KUKA KRL program: EPS_2_25748_MH03A_A_20260121065858.src

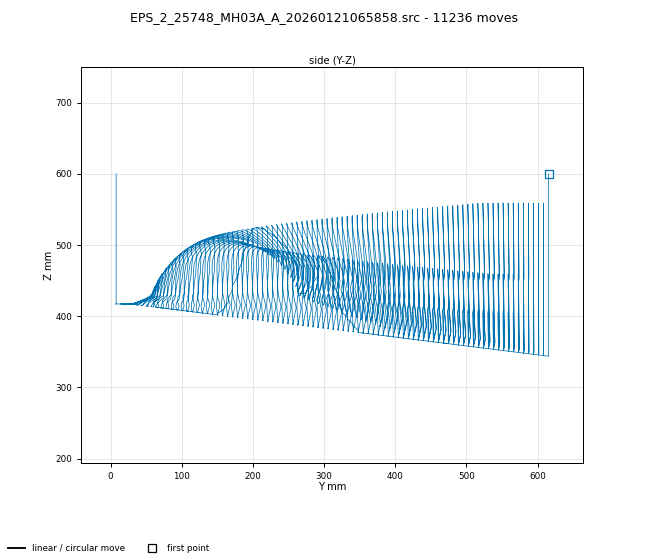
[picture p0: tool path of EPS_2_25748_MH03A_A_20260121065858.src, 11236 of 11238 moves have a stored position in this frame; points joined in program order, loops and branches not executed]
&ACCESS RVP
&REL 4
&COMMENT QRS 19112012
&PARAM EDITMASK = *
DEF PART()
EXT BAS (BAS_COMMAND :IN,REAL :IN )
INT I
BAS (#INITMOV,0 )

;KUKA QRS Post kuka4.cps  Date:22-06-2017 !

File_ID=2998

QRS_PRE_INIT()

;Init var - Until changes are made in qrs_pre_init
Outlet_Square_prg=0
Inlet_1_Square_prg=0
Inlet_2_Square_prg=0
Inlet_3_Square_prg=0
Inlet_4_Square_prg=0
Inlet_5_Square_prg=0

Outlet_1={X 0.000, Y 520.860, Z 458.500, B 0.000, E1 0.000 }
Inlet_1={X 0.000, Y 535.970, Z 408.500, B 0.000, E1 270.000 }
Outlet_1_type=201
Inlet_1_type=101
;QRS#1=Sidecore dimensions
;QRS#2=200-8" PVC SDR 35
;QRS#3=100-4" PVC SDR 28
;QRS#4=
;QRS#5=
;QRS#6=
;QRS#7=
;QRS#8=
;QRS#9=12-08 PSX
;QRS#10=8QRS PSX
;QRS#11=
;QRS#12=
;QRS#13=
;QRS#14=
;QRS#15=
;QRS#16=1220x127x838 2,75'
;QRS#17=EPS Height
;QRS#18=559
;QRS#19=*
;QRS#20= UPDATED VERSION 22-06-2017
;QRS#21=*
Outlet_Square=0100
Inlet_1_Square=045
Inlet_2_Square=0
Inlet_3_Square=0
Inlet_4_Square=0
Inlet_5_Square=0
Mill_Square=1
Outlet_Square_Prg=204
Inlet_1_Square_prg=201

QRS_INIT()

$ADVANCE=5

; T1
PTP {E1 173.608,E2 173.608}
PTP {X 0,Y 615.501,A -85,B 0,C 180,E1 173.608,E2 173.608,E3 0,E4 0,E5 0,E6 0}
QRS_SPEED_INIT()
LIN {X 0,Y 615.501,Z 600,A -85,B 0,C 180,E1 173.608,E2 173.608,E3 0,E4 0,E5 0,E6 0} C_VEL
LIN {X 0,Y 615.501,Z 353.868,A -85,B 0,C 180,E1 173.608,E2 173.608} C_VEL
LIN {X 0,Y 615.501,Z 345.693,A -85,B 0,C 180,E1 173.608,E2 173.608} C_VEL
LIN {X 0,Y 615.488,Z 343.693,A -85,B 0,C 180,E1 173.422,E2 173.422} C_VEL
LIN {X 0,Y 615.492,Z 343.688,A -85,B 0,C 180,E1 170.801,E2 170.801} C_VEL
LIN {X 0,Y 615.492,Z 343.699,A -85,B 0,C 180,E1 168.139,E2 168.139} C_VEL
LIN {X 0,Y 615.481,Z 343.69,A -85,B 0,C 180,E1 165.451,E2 165.451} C_VEL
LIN {X 0,Y 615.493,Z 343.692,A -85,B 0,C 180,E1 162.73,E2 162.73} C_VEL
LIN {X 0,Y 615.49,Z 343.695,A -85,B 0,C 180,E1 159.967,E2 159.967} C_VEL
LIN {X 0,Y 615.481,Z 343.69,A -85,B 0,C 180,E1 157.155,E2 157.155} C_VEL
LIN {X 0,Y 615.482,Z 343.693,A -85,B 0,C 180,E1 154.284,E2 154.284} C_VEL
LIN {X 0,Y 615.479,Z 343.699,A -85,B 0,C 180,E1 151.551,E2 151.551} C_VEL
LIN {X 0,Y 615.485,Z 343.689,A -85,B 0,C 180,E1 148.915,E2 148.915} C_VEL
LIN {X 0,Y 615.49,Z 343.692,A -85,B 0,C 180,E1 145.978,E2 145.978} C_VEL
LIN {X 0,Y 615.487,Z 343.702,A -85,B 0,C 180,E1 143.063,E2 143.063} C_VEL
LIN {X 0,Y 615.49,Z 343.689,A -85,B 0,C 180,E1 140.25,E2 140.25} C_VEL
LIN {X 0,Y 615.485,Z 343.693,A -85,B 0,C 180,E1 137.647,E2 137.647} C_VEL
LIN {X 0,Y 615.491,Z 343.694,A -85,B 0,C 180,E1 134.932,E2 134.932} C_VEL
LIN {X 0,Y 615.485,Z 343.689,A -85,B 0,C 180,E1 132.08,E2 132.08} C_VEL
LIN {X 0,Y 615.489,Z 343.7,A -85,B 0,C 180,E1 129.75,E2 129.75} C_VEL
LIN {X 0,Y 615.476,Z 343.692,A -85,B 0,C 180,E1 126.935,E2 126.935} C_VEL
LIN {X 0,Y 615.492,Z 343.701,A -85,B 0,C 180,E1 124.701,E2 124.701} C_VEL
LIN {X 0,Y 615.49,Z 343.688,A -85,B 0,C 180,E1 122.331,E2 122.331} C_VEL
LIN {X 0,Y 615.492,Z 343.695,A -85,B 0,C 180,E1 119.406,E2 119.406} C_VEL
LIN {X 0,Y 615.476,Z 343.691,A -85,B 0,C 180,E1 117.042,E2 117.042} C_VEL
LIN {X 0,Y 615.48,Z 343.694,A -85,B 0,C 180,E1 114.272,E2 114.272} C_VEL
LIN {X 0,Y 615.496,Z 343.697,A -85,B 0,C 180,E1 111.431,E2 111.431} C_VEL
LIN {X 0,Y 615.488,Z 343.689,A -85,B 0,C 180,E1 108.604,E2 108.604} C_VEL
LIN {X 0,Y 615.492,Z 343.691,A -85,B 0,C 180,E1 105.905,E2 105.905} C_VEL
LIN {X 0,Y 615.485,Z 343.696,A -85,B 0,C 180,E1 103.201,E2 103.201} C_VEL
LIN {X 0,Y 615.481,Z 343.69,A -85,B 0,C 180,E1 100.527,E2 100.527} C_VEL
LIN {X 0,Y 615.487,Z 343.701,A -85,B 0,C 180,E1 97.876,E2 97.876} C_VEL
LIN {X 0,Y 615.48,Z 343.691,A -85,B 0,C 180,E1 95.241,E2 95.241} C_VEL
LIN {X 0,Y 615.48,Z 343.695,A -85,B 0,C 180,E1 92.618,E2 92.618} C_VEL
LIN {X 0,Y 615.49,Z 343.692,A -85,B 0,C 180,E1 90,E2 90} C_VEL
LIN {X 0,Y 615.48,Z 343.692,A -85,B 0,C 180,E1 87.382,E2 87.382} C_VEL
LIN {X 0,Y 615.486,Z 343.698,A -85,B 0,C 180,E1 84.759,E2 84.759} C_VEL
LIN {X 0,Y 615.488,Z 343.688,A -85,B 0,C 180,E1 82.124,E2 82.124} C_VEL
LIN {X 0,Y 615.497,Z 343.697,A -85,B 0,C 180,E1 79.473,E2 79.473} C_VEL
LIN {X 0,Y 615.479,Z 343.692,A -85,B 0,C 180,E1 76.798,E2 76.798} C_VEL
LIN {X 0,Y 615.485,Z 343.691,A -85,B 0,C 180,E1 74.095,E2 74.095} C_VEL
LIN {X 0,Y 615.488,Z 343.699,A -85,B 0,C 180,E1 71.354,E2 71.354} C_VEL
LIN {X 0,Y 615.485,Z 343.689,A -85,B 0,C 180,E1 68.568,E2 68.568} C_VEL
LIN {X 0,Y 615.482,Z 343.692,A -85,B 0,C 180,E1 65.728,E2 65.728} C_VEL
LIN {X 0,Y 615.492,Z 343.7,A -85,B 0,C 180,E1 62.955,E2 62.955} C_VEL
LIN {X 0,Y 615.482,Z 343.69,A -85,B 0,C 180,E1 60.207,E2 60.207} C_VEL
LIN {X 0,Y 615.495,Z 343.692,A -85,B 0,C 180,E1 57.543,E2 57.543} C_VEL
LIN {X 0,Y 615.478,Z 343.691,A -85,B 0,C 180,E1 55.184,E2 55.184} C_VEL
LIN {X 0,Y 615.497,Z 343.697,A -85,B 0,C 180,E1 52.758,E2 52.758} C_VEL
LIN {X 0,Y 615.482,Z 343.694,A -85,B 0,C 180,E1 49.912,E2 49.912} C_VEL
LIN {X 0,Y 615.495,Z 343.695,A -85,B 0,C 180,E1 47.647,E2 47.647} C_VEL
LIN {X 0,Y 615.482,Z 343.693,A -85,B 0,C 180,E1 44.931,E2 44.931} C_VEL
LIN {X 0,Y 615.482,Z 343.69,A -85,B 0,C 180,E1 42.079,E2 42.079} C_VEL
LIN {X 0,Y 615.496,Z 343.694,A -85,B 0,C 180,E1 39.75,E2 39.75} C_VEL
LIN {X 0,Y 615.486,Z 343.689,A -85,B 0,C 180,E1 36.936,E2 36.936} C_VEL
LIN {X 0,Y 615.487,Z 343.691,A -85,B 0,C 180,E1 34.022,E2 34.022} C_VEL
LIN {X 0,Y 615.49,Z 343.699,A -85,B 0,C 180,E1 31.086,E2 31.086} C_VEL
LIN {X 0,Y 615.489,Z 343.835,A -85,B 0,C 180,E1 29.697,E2 29.697} C_VEL
LIN {X 0,Y 615.498,Z 350.25,A -85,B 0,C 180,E1 27.046,E2 27.046} C_VEL
LIN {X 0,Y 615.488,Z 357.77,A -85,B 0,C 180,E1 24.008,E2 24.008} C_VEL
LIN {X 0,Y 615.478,Z 364.29,A -85,B 0,C 180,E1 21.432,E2 21.432} C_VEL
LIN {X 0,Y 615.476,Z 371.461,A -85,B 0,C 180,E1 18.646,E2 18.646} C_VEL
LIN {X 0,Y 615.488,Z 378.635,A -85,B 0,C 180,E1 15.905,E2 15.905} C_VEL
LIN {X 0,Y 615.494,Z 385.799,A -85,B 0,C 180,E1 13.201,E2 13.201} C_VEL
LIN {X 0,Y 615.486,Z 392.972,A -85,B 0,C 180,E1 10.527,E2 10.527} C_VEL
LIN {X 0,Y 615.478,Z 400.129,A -85,B 0,C 180,E1 7.876,E2 7.876} C_VEL
LIN {X 0,Y 615.487,Z 403.222,A -85,B 0,C 180,E1 6.737,E2 6.737} C_VEL
LIN {X 0,Y 615.489,Z 413.526,A -85,B 0,C 180,E1 6.392,E2 6.392} C_VEL
LIN {X 0,Y 615.478,Z 421.945,A -85,B 0,C 180,E1 5.981,E2 5.981} C_VEL
LIN {X 0,Y 615.487,Z 429.67,A -85,B 0,C 180,E1 5.488,E2 5.488} C_VEL
LIN {X 0,Y 615.489,Z 436.516,A -85,B 0,C 180,E1 4.913,E2 4.913} C_VEL
LIN {X 0,Y 615.497,Z 442.667,A -85,B 0,C 180,E1 4.256,E2 4.256} C_VEL
LIN {X 0,Y 615.497,Z 447.515,A -85,B 0,C 180,E1 3.601,E2 3.601} C_VEL
LIN {X 0,Y 615.496,Z 451.25,A -85,B 0,C 180,E1 2.945,E2 2.945} C_VEL
LIN {X 0,Y 615.498,Z 455.229,A -85,B 0,C 180,E1 1.963,E2 1.963} C_VEL
LIN {X 0,Y 615.497,Z 456.963,A -85,B 0,C 180,E1 1.309,E2 1.309} C_VEL
LIN {X 0,Y 615.496,Z 458.004,A -85,B 0,C 180,E1 0.654,E2 0.654} C_VEL
LIN {X 0,Y 615.494,Z 458.384,A -85,B 0,C 180,E1 0,E2 0} C_VEL
LIN {X 0,Y 615.496,Z 458.105,A -85,B 0,C 180,E1 -0.654,E2 -0.654} C_VEL
LIN {X 0,Y 615.497,Z 457.166,A -85,B 0,C 180,E1 -1.309,E2 -1.309} C_VEL
LIN {X 0,Y 615.496,Z 455.536,A -85,B 0,C 180,E1 -1.963,E2 -1.963} C_VEL
LIN {X 0,Y 615.498,Z 451.663,A -85,B 0,C 180,E1 -2.945,E2 -2.945} C_VEL
LIN {X 0,Y 615.5,Z 447.012,A -85,B 0,C 180,E1 -3.764,E2 -3.764} C_VEL
LIN {X 0,Y 615.498,Z 442.03,A -85,B 0,C 180,E1 -4.42,E2 -4.42} C_VEL
LIN {X 0,Y 615.482,Z 435.756,A -85,B 0,C 180,E1 -5.077,E2 -5.077} C_VEL
LIN {X 0,Y 615.483,Z 428.589,A -85,B 0,C 180,E1 -5.652,E2 -5.652} C_VEL
LIN {X 0,Y 615.483,Z 420.605,A -85,B 0,C 180,E1 -6.145,E2 -6.145} C_VEL
LIN {X 0,Y 615.492,Z 411.022,A -85,B 0,C 180,E1 -6.579,E2 -6.579} C_VEL
LIN {X 0,Y 615.48,Z 403.195,A -85,B 0,C 180,E1 -6.838,E2 -6.838} C_VEL
LIN {X 0,Y 615.489,Z 396.799,A -85,B 0,C 180,E1 -9.199,E2 -9.199} C_VEL
LIN {X 0,Y 615.477,Z 389.625,A -85,B 0,C 180,E1 -11.861,E2 -11.861} C_VEL
LIN {X 0,Y 615.481,Z 382.466,A -85,B 0,C 180,E1 -14.549,E2 -14.549} C_VEL
LIN {X 0,Y 615.492,Z 375.279,A -85,B 0,C 180,E1 -17.27,E2 -17.27} C_VEL
LIN {X 0,Y 615.493,Z 368.112,A -85,B 0,C 180,E1 -20.033,E2 -20.033} C_VEL
LIN {X 0,Y 615.482,Z 360.924,A -85,B 0,C 180,E1 -22.845,E2 -22.845} C_VEL
LIN {X 0,Y 615.476,Z 354.12,A -85,B 0,C 180,E1 -25.566,E2 -25.566} C_VEL
LIN {X 0,Y 615.485,Z 348.349,A -85,B 0,C 180,E1 -27.915,E2 -27.915} C_VEL
LIN {X 0,Y 615.494,Z 343.696,A -85,B 0,C 180,E1 -29.886,E2 -29.886} C_VEL
LIN {X 0,Y 615.487,Z 343.699,A -85,B 0,C 180,E1 -32.458,E2 -32.458} C_VEL
LIN {X 0,Y 615.498,Z 343.7,A -85,B 0,C 180,E1 -34.815,E2 -34.815} C_VEL
LIN {X 0,Y 615.481,Z 343.699,A -85,B 0,C 180,E1 -37.243,E2 -37.243} C_VEL
LIN {X 0,Y 615.497,Z 343.7,A -85,B 0,C 180,E1 -40.09,E2 -40.09} C_VEL
LIN {X 0,Y 615.491,Z 343.699,A -85,B 0,C 180,E1 -43.047,E2 -43.047} C_VEL
LIN {X 0,Y 615.491,Z 343.697,A -85,B 0,C 180,E1 -46.002,E2 -46.002} C_VEL
LIN {X 0,Y 615.497,Z 343.7,A -85,B 0,C 180,E1 -48.527,E2 -48.527} C_VEL
LIN {X 0,Y 615.478,Z 343.699,A -85,B 0,C 180,E1 -51.095,E2 -51.095} C_VEL
LIN {X 0,Y 615.491,Z 343.699,A -85,B 0,C 180,E1 -53.575,E2 -53.575} C_VEL
LIN {X 0,Y 615.493,Z 343.696,A -85,B 0,C 180,E1 -56.465,E2 -56.465} C_VEL
LIN {X 0,Y 615.491,Z 343.7,A -85,B 0,C 180,E1 -59.08,E2 -59.08} C_VEL
LIN {X 0,Y 615.494,Z 343.696,A -85,B 0,C 180,E1 -61.549,E2 -61.549} C_VEL
LIN {X 0,Y 615.488,Z 343.839,A -85,B 0,C 180,E1 -62.593,E2 -62.593} C_VEL
LIN {X 0,Y 615.489,Z 361.436,A -85,B 0,C 180,E1 -65.369,E2 -65.369} C_VEL
LIN {X 0,Y 615.488,Z 379.892,A -85,B 0,C 180,E1 -68.216,E2 -68.216} C_VEL
LIN {X 0,Y 615.492,Z 398.326,A -85,B 0,C 180,E1 -71.008,E2 -71.008} C_VEL
LIN {X 0,Y 615.493,Z 417.271,A -85,B 0,C 180,E1 -73.832,E2 -73.832} C_VEL
LIN {X 0,Y 615.478,Z 436.29,A -85,B 0,C 180,E1 -76.63,E2 -76.63} C_VEL
LIN {X 0,Y 615.497,Z 447.777,A -85,B 0,C 180,E1 -78.306,E2 -78.306} C_VEL
LIN {X 0,Y 615.483,Z 462.234,A -85,B 0,C 180,E1 -78.556,E2 -78.556} C_VEL
LIN {X 0,Y 615.481,Z 475.31,A -85,B 0,C 180,E1 -78.921,E2 -78.921} C_VEL
LIN {X 0,Y 615.489,Z 487.115,A -85,B 0,C 180,E1 -79.383,E2 -79.383} C_VEL
LIN {X 0,Y 615.487,Z 498.572,A -85,B 0,C 180,E1 -79.972,E2 -79.972} C_VEL
LIN {X 0,Y 615.499,Z 510.019,A -85,B 0,C 180,E1 -80.718,E2 -80.718} C_VEL
LIN {X 0,Y 615.498,Z 519.255,A -85,B 0,C 180,E1 -81.463,E2 -81.463} C_VEL
LIN {X 0,Y 615.499,Z 527.652,A -85,B 0,C 180,E1 -82.289,E2 -82.289} C_VEL
LIN {X 0,Y 615.497,Z 535.69,A -85,B 0,C 180,E1 -83.259,E2 -83.259} C_VEL
LIN {X 0,Y 615.499,Z 541.422,A -85,B 0,C 180,E1 -84.101,E2 -84.101} C_VEL
LIN {X 0,Y 615.496,Z 546.872,A -85,B 0,C 180,E1 -85.087,E2 -85.087} C_VEL
LIN {X 0,Y 615.496,Z 551.14,A -85,B 0,C 180,E1 -86.071,E2 -86.071} C_VEL
LIN {X 0,Y 615.495,Z 553.398,A -85,B 0,C 180,E1 -86.727,E2 -86.727} C_VEL
LIN {X 0,Y 615.497,Z 555.233,A -85,B 0,C 180,E1 -87.382,E2 -87.382} C_VEL
LIN {X 0,Y 615.499,Z 556.607,A -85,B 0,C 180,E1 -88.037,E2 -88.037} C_VEL
LIN {X 0,Y 615.496,Z 558.173,A -85,B 0,C 180,E1 -89.346,E2 -89.346} C_VEL
LIN {X 0,Y 615.494,Z 558.389,A -85,B 0,C 180,E1 -90,E2 -90} C_VEL
LIN {X 0,Y 615.496,Z 557.58,A -85,B 0,C 180,E1 -91.308,E2 -91.308} C_VEL
LIN {X 0,Y 615.499,Z 556.608,A -85,B 0,C 180,E1 -91.963,E2 -91.963} C_VEL
LIN {X 0,Y 615.497,Z 555.233,A -85,B 0,C 180,E1 -92.618,E2 -92.618} C_VEL
LIN {X 0,Y 615.496,Z 552.35,A -85,B 0,C 180,E1 -93.601,E2 -93.601} C_VEL
LIN {X 0,Y 615.498,Z 548.442,A -85,B 0,C 180,E1 -94.584,E2 -94.584} C_VEL
LIN {X 0,Y 615.499,Z 543.405,A -85,B 0,C 180,E1 -95.57,E2 -95.57} C_VEL
LIN {X 0,Y 615.497,Z 536.87,A -85,B 0,C 180,E1 -96.583,E2 -96.583} C_VEL
LIN {X 0,Y 615.497,Z 529.134,A -85,B 0,C 180,E1 -97.545,E2 -97.545} C_VEL
LIN {X 0,Y 615.498,Z 521.046,A -85,B 0,C 180,E1 -98.371,E2 -98.371} C_VEL
LIN {X 0,Y 615.499,Z 511.169,A -85,B 0,C 180,E1 -99.199,E2 -99.199} C_VEL
LIN {X 0,Y 615.492,Z 499.982,A -85,B 0,C 180,E1 -99.945,E2 -99.945} C_VEL
LIN {X 0,Y 615.484,Z 489.025,A -85,B 0,C 180,E1 -100.527,E2 -100.527} C_VEL
LIN {X 0,Y 615.482,Z 476.477,A -85,B 0,C 180,E1 -101.041,E2 -101.041} C_VEL
LIN {X 0,Y 615.481,Z 464.07,A -85,B 0,C 180,E1 -101.402,E2 -101.402} C_VEL
LIN {X 0,Y 615.495,Z 450.47,A -85,B 0,C 180,E1 -101.652,E2 -101.652} C_VEL
LIN {X 0,Y 615.497,Z 447.778,A -85,B 0,C 180,E1 -101.693,E2 -101.693} C_VEL
LIN {X 0,Y 615.494,Z 427.094,A -85,B 0,C 180,E1 -104.718,E2 -104.718} C_VEL
LIN {X 0,Y 615.492,Z 407.539,A -85,B 0,C 180,E1 -107.613,E2 -107.613} C_VEL
LIN {X 0,Y 615.487,Z 389.682,A -85,B 0,C 180,E1 -110.295,E2 -110.295} C_VEL
LIN {X 0,Y 615.479,Z 371.822,A -85,B 0,C 180,E1 -113.022,E2 -113.022} C_VEL
LIN {X 0,Y 615.5,Z 354.515,A -85,B 0,C 180,E1 -115.715,E2 -115.715} C_VEL
LIN {X 0,Y 615.489,Z 343.689,A -85,B 0,C 180,E1 -117.453,E2 -117.453} C_VEL
LIN {X 0,Y 615.5,Z 343.7,A -85,B 0,C 180,E1 -120.159,E2 -120.159} C_VEL
LIN {X 0,Y 615.494,Z 343.688,A -85,B 0,C 180,E1 -122.457,E2 -122.457} C_VEL
LIN {X 0,Y 615.487,Z 343.693,A -85,B 0,C 180,E1 -124.815,E2 -124.815} C_VEL
LIN {X 0,Y 615.487,Z 343.692,A -85,B 0,C 180,E1 -127.242,E2 -127.242} C_VEL
LIN {X 0,Y 615.492,Z 343.699,A -85,B 0,C 180,E1 -130.089,E2 -130.089} C_VEL
LIN {X 0,Y 615.495,Z 343.689,A -85,B 0,C 180,E1 -132.352,E2 -132.352} C_VEL
LIN {X 0,Y 615.489,Z 343.699,A -85,B 0,C 180,E1 -135.068,E2 -135.068} C_VEL
LIN {X 0,Y 615.482,Z 343.691,A -85,B 0,C 180,E1 -137.92,E2 -137.92} C_VEL
LIN {X 0,Y 615.491,Z 343.7,A -85,B 0,C 180,E1 -140.25,E2 -140.25} C_VEL
LIN {X 0,Y 615.488,Z 343.691,A -85,B 0,C 180,E1 -143.063,E2 -143.063} C_VEL
LIN {X 0,Y 615.489,Z 343.688,A -85,B 0,C 180,E1 -145.978,E2 -145.978} C_VEL
LIN {X 0,Y 615.482,Z 343.694,A -85,B 0,C 180,E1 -148.915,E2 -148.915} C_VEL
LIN {X 0,Y 615.48,Z 343.695,A -85,B 0,C 180,E1 -151.551,E2 -151.551} C_VEL
LIN {X 0,Y 615.478,Z 343.69,A -85,B 0,C 180,E1 -154.284,E2 -154.284} C_VEL
LIN {X 0,Y 615.476,Z 343.694,A -85,B 0,C 180,E1 -156.443,E2 -156.443} C_VEL
LIN {X 0,Y 615.499,Z 343.699,A -85,B 0,C 180,E1 -158.568,E2 -158.568} C_VEL
LIN {X 0,Y 615.477,Z 343.693,A -85,B 0,C 180,E1 -161.398,E2 -161.398} C_VEL
LIN {X 0,Y 615.478,Z 343.692,A -85,B 0,C 180,E1 -164.095,E2 -164.095} C_VEL
LIN {X 0,Y 615.498,Z 343.697,A -85,B 0,C 180,E1 -166.799,E2 -166.799} C_VEL
LIN {X 0,Y 615.486,Z 343.689,A -85,B 0,C 180,E1 -169.473,E2 -169.473} C_VEL
LIN {X 0,Y 615.484,Z 343.697,A -85,B 0,C 180,E1 -172.124,E2 -172.124} C_VEL
LIN {X 0,Y 615.487,Z 343.691,A -85,B 0,C 180,E1 -174.759,E2 -174.759} C_VEL
LIN {X 0,Y 615.492,Z 343.69,A -85,B 0,C 180,E1 -177.382,E2 -177.382} C_VEL
LIN {X 0,Y 615.489,Z 343.695,A -85,B 0,C 180,E1 -180,E2 -180} C_VEL
LIN {X 0,Y 615.488,Z 343.688,A -85,B 0,C 180,E1 -182.618,E2 -182.618} C_VEL
LIN {X 0,Y 615.496,Z 343.7,A -85,B 0,C 180,E1 -185.241,E2 -185.241} C_VEL
LIN {X 0,Y 615.488,Z 343.693,A -85,B 0,C 180,E1 -186.578,E2 -186.578} C_VEL
LIN {X 0,Y 614.817,Z 343.842,A -85,B 0,C 180,E1 -187.124,E2 -187.124} C_VEL
LIN {X 0,Y 611.986,Z 344.251,A -85,B 0,C 180,E1 -188.01,E2 -188.01} C_VEL
LIN {X 0,Y 609.592,Z 344.56,A -85,B 0,C 180,E1 -188.723,E2 -188.723} C_VEL
LIN {X 0,Y 608.553,Z 344.679,A -85,B 0,C 180,E1 -189.272,E2 -189.272} C_VEL
LIN {X 0,Y 608.461,Z 344.689,A -85,B 0,C 180,E1 -189.459,E2 -189.459} C_VEL
LIN {X 0,Y 608.466,Z 344.696,A -85,B 0,C 180,E1 -192,E2 -192} C_VEL
LIN {X 0,Y 608.472,Z 344.689,A -85,B 0,C 180,E1 -194.721,E2 -194.721} C_VEL
LIN {X 0,Y 608.456,Z 344.691,A -85,B 0,C 180,E1 -197.477,E2 -197.477} C_VEL
LIN {X 0,Y 608.464,Z 344.697,A -85,B 0,C 180,E1 -200.274,E2 -200.274} C_VEL
LIN {X 0,Y 608.46,Z 344.691,A -85,B 0,C 180,E1 -202.476,E2 -202.476} C_VEL
LIN {X 0,Y 608.457,Z 344.69,A -85,B 0,C 180,E1 -204.571,E2 -204.571} C_VEL
LIN {X 0,Y 608.484,Z 344.69,A -85,B 0,C 180,E1 -207.208,E2 -207.208} C_VEL
LIN {X 0,Y 608.47,Z 344.691,A -85,B 0,C 180,E1 -209.972,E2 -209.972} C_VEL
LIN {X 0,Y 608.455,Z 344.69,A -85,B 0,C 180,E1 -212.88,E2 -212.88} C_VEL
LIN {X 0,Y 608.443,Z 344.699,A -85,B 0,C 180,E1 -215.278,E2 -215.278} C_VEL
LIN {X 0,Y 608.466,Z 344.689,A -85,B 0,C 180,E1 -217.747,E2 -217.747} C_VEL
LIN {X 0,Y 608.453,Z 344.698,A -85,B 0,C 180,E1 -220.329,E2 -220.329} C_VEL
LIN {X 0,Y 608.452,Z 344.691,A -85,B 0,C 180,E1 -222.96,E2 -222.96} C_VEL
LIN {X 0,Y 608.46,Z 344.692,A -85,B 0,C 180,E1 -225.736,E2 -225.736} C_VEL
LIN {X 0,Y 608.462,Z 344.697,A -85,B 0,C 180,E1 -228.658,E2 -228.658} C_VEL
LIN {X 0,Y 608.471,Z 344.692,A -85,B 0,C 180,E1 -231.76,E2 -231.76} C_VEL
LIN {X 0,Y 608.448,Z 344.695,A -85,B 0,C 180,E1 -233.955,E2 -233.955} C_VEL
LIN {X 0,Y 608.465,Z 344.689,A -85,B 0,C 180,E1 -236.329,E2 -236.329} C_VEL
LIN {X 0,Y 608.449,Z 344.698,A -85,B 0,C 180,E1 -238.733,E2 -238.733} C_VEL
LIN {X 0,Y 608.473,Z 344.688,A -85,B 0,C 180,E1 -241.38,E2 -241.38} C_VEL
LIN {X 0,Y 608.478,Z 344.688,A -85,B 0,C 180,E1 -244.278,E2 -244.278} C_VEL
LIN {X 0,Y 608.455,Z 344.696,A -85,B 0,C 180,E1 -246.876,E2 -246.876} C_VEL
LIN {X 0,Y 608.468,Z 344.689,A -85,B 0,C 180,E1 -249.322,E2 -249.322} C_VEL
LIN {X 0,Y 608.456,Z 344.695,A -85,B 0,C 180,E1 -251.828,E2 -251.828} C_VEL
LIN {X 0,Y 608.467,Z 344.689,A -85,B 0,C 180,E1 -254.594,E2 -254.594} C_VEL
LIN {X 0,Y 608.473,Z 344.691,A -85,B 0,C 180,E1 -257.323,E2 -257.323} C_VEL
LIN {X 0,Y 608.465,Z 344.692,A -85,B 0,C 180,E1 -260.023,E2 -260.023} C_VEL
LIN {X 0,Y 608.462,Z 344.69,A -85,B 0,C 180,E1 -262.701,E2 -262.701} C_VEL
LIN {X 0,Y 608.464,Z 344.697,A -85,B 0,C 180,E1 -265.363,E2 -265.363} C_VEL
LIN {X 0,Y 608.469,Z 344.689,A -85,B 0,C 180,E1 -268.014,E2 -268.014} C_VEL
LIN {X 0,Y 608.48,Z 344.691,A -85,B 0,C 180,E1 -270.662,E2 -270.662} C_VEL
LIN {X 0,Y 608.475,Z 344.69,A -85,B 0,C 180,E1 -273.311,E2 -273.311} C_VEL
LIN {X 0,Y 608.492,Z 344.686,A -85,B 0,C 180,E1 -275.967,E2 -275.967} C_VEL
LIN {X 0,Y 608.457,Z 344.696,A -85,B 0,C 180,E1 -278.636,E2 -278.636} C_VEL
LIN {X 0,Y 608.459,Z 344.69,A -85,B 0,C 180,E1 -281.324,E2 -281.324} C_VEL
LIN {X 0,Y 608.473,Z 344.691,A -85,B 0,C 180,E1 -284.038,E2 -284.038} C_VEL
LIN {X 0,Y 608.479,Z 344.69,A -85,B 0,C 180,E1 -286.783,E2 -286.783} C_VEL
LIN {X 0,Y 608.45,Z 344.691,A -85,B 0,C 180,E1 -289.571,E2 -289.571} C_VEL
LIN {X 0,Y 608.481,Z 344.69,A -85,B 0,C 180,E1 -292.405,E2 -292.405} C_VEL
LIN {X 0,Y 608.454,Z 344.696,A -85,B 0,C 180,E1 -295.301,E2 -295.301} C_VEL
LIN {X 0,Y 608.451,Z 344.693,A -85,B 0,C 180,E1 -297.518,E2 -297.518} C_VEL
LIN {X 0,Y 608.463,Z 344.691,A -85,B 0,C 180,E1 -299.97,E2 -299.97} C_VEL
LIN {X 0,Y 608.461,Z 344.689,A -85,B 0,C 180,E1 -302.88,E2 -302.88} C_VEL
LIN {X 0,Y 608.44,Z 344.697,A -85,B 0,C 180,E1 -305.278,E2 -305.278} C_VEL
LIN {X 0,Y 608.469,Z 344.689,A -85,B 0,C 180,E1 -307.747,E2 -307.747} C_VEL
LIN {X 0,Y 608.451,Z 344.696,A -85,B 0,C 180,E1 -310.329,E2 -310.329} C_VEL
LIN {X 0,Y 608.452,Z 344.691,A -85,B 0,C 180,E1 -312.96,E2 -312.96} C_VEL
LIN {X 0,Y 608.45,Z 344.695,A -85,B 0,C 180,E1 -315.737,E2 -315.737} C_VEL
LIN {X 0,Y 608.46,Z 344.695,A -85,B 0,C 180,E1 -318.658,E2 -318.658} C_VEL
LIN {X 0,Y 608.472,Z 344.688,A -85,B 0,C 180,E1 -321.412,E2 -321.412} C_VEL
LIN {X 0,Y 608.482,Z 344.693,A -85,B 0,C 180,E1 -323.95,E2 -323.95} C_VEL
LIN {X 0,Y 608.448,Z 344.691,A -85,B 0,C 180,E1 -326.328,E2 -326.328} C_VEL
LIN {X 0,Y 608.465,Z 344.695,A -85,B 0,C 180,E1 -328.73,E2 -328.73} C_VEL
LIN {X 0,Y 608.481,Z 344.879,A -85,B 0,C 180,E1 -330.316,E2 -330.316} C_VEL
LIN {X 0,Y 608.446,Z 351.891,A -85,B 0,C 180,E1 -333.225,E2 -333.225} C_VEL
LIN {X 0,Y 608.457,Z 358.354,A -85,B 0,C 180,E1 -335.853,E2 -335.853} C_VEL
LIN {X 0,Y 608.442,Z 364.518,A -85,B 0,C 180,E1 -338.307,E2 -338.307} C_VEL
LIN {X 0,Y 608.431,Z 371.734,A -85,B 0,C 180,E1 -341.13,E2 -341.13} C_VEL
LIN {X 0,Y 608.446,Z 378.949,A -85,B 0,C 180,E1 -343.906,E2 -343.906} C_VEL
LIN {X 0,Y 608.437,Z 386.166,A -85,B 0,C 180,E1 -346.643,E2 -346.643} C_VEL
LIN {X 0,Y 608.424,Z 393.382,A -85,B 0,C 180,E1 -349.349,E2 -349.349} C_VEL
LIN {X 0,Y 608.41,Z 400.599,A -85,B 0,C 180,E1 -352.032,E2 -352.032} C_VEL
LIN {X 0,Y 608.433,Z 403.853,A -85,B 0,C 180,E1 -353.186,E2 -353.186} C_VEL
LIN {X 0,Y 608.478,Z 414.079,A -85,B 0,C 180,E1 -353.534,E2 -353.534} C_VEL
LIN {X 0,Y 608.454,Z 422.472,A -85,B 0,C 180,E1 -353.95,E2 -353.95} C_VEL
LIN {X 0,Y 608.453,Z 431.252,A -85,B 0,C 180,E1 -354.532,E2 -354.532} C_VEL
LIN {X 0,Y 608.448,Z 437.027,A -85,B 0,C 180,E1 -355.03,E2 -355.03} C_VEL
LIN {X 0,Y 608.443,Z 443.205,A -85,B 0,C 180,E1 -355.694,E2 -355.694} C_VEL
LIN {X 0,Y 608.451,Z 448.067,A -85,B 0,C 180,E1 -356.358,E2 -356.358} C_VEL
LIN {X 0,Y 608.451,Z 451.818,A -85,B 0,C 180,E1 -357.021,E2 -357.021} C_VEL
LIN {X 0,Y 608.443,Z 455.825,A -85,B 0,C 180,E1 -358.014,E2 -358.014} C_VEL
LIN {X 0,Y 608.449,Z 457.568,A -85,B 0,C 180,E1 -358.676,E2 -358.676} C_VEL
LIN {X 0,Y 608.439,Z 458.615,A -85,B 0,C 180,E1 -359.338,E2 -359.338} C_VEL
LIN {X 0,Y 608.434,Z 458.995,A -85,B 0,C 180,E1 -360,E2 -360} C_VEL
LIN {X 0,Y 608.439,Z 458.714,A -85,B 0,C 180,E1 -360.662,E2 -360.662} C_VEL
LIN {X 0,Y 608.449,Z 457.768,A -85,B 0,C 180,E1 -361.324,E2 -361.324} C_VEL
LIN {X 0,Y 608.442,Z 456.128,A -85,B 0,C 180,E1 -361.986,E2 -361.986} C_VEL
LIN {X 0,Y 608.429,Z 453.745,A -85,B 0,C 180,E1 -362.648,E2 -362.648} C_VEL
LIN {X 0,Y 608.452,Z 448.618,A -85,B 0,C 180,E1 -363.642,E2 -363.642} C_VEL
LIN {X 0,Y 608.451,Z 442.555,A -85,B 0,C 180,E1 -364.472,E2 -364.472} C_VEL
LIN {X 0,Y 608.433,Z 436.249,A -85,B 0,C 180,E1 -365.136,E2 -365.136} C_VEL
LIN {X 0,Y 608.458,Z 429.093,A -85,B 0,C 180,E1 -365.717,E2 -365.717} C_VEL
LIN {X 0,Y 608.443,Z 421.107,A -85,B 0,C 180,E1 -366.217,E2 -366.217} C_VEL
LIN {X 0,Y 608.483,Z 412.26,A -85,B 0,C 180,E1 -366.632,E2 -366.632} C_VEL
LIN {X 0,Y 608.426,Z 403.694,A -85,B 0,C 180,E1 -366.913,E2 -366.913} C_VEL
LIN {X 0,Y 608.418,Z 397.233,A -85,B 0,C 180,E1 -369.307,E2 -369.307} C_VEL
LIN {X 0,Y 608.418,Z 390.014,A -85,B 0,C 180,E1 -372.001,E2 -372.001} C_VEL
LIN {X 0,Y 608.441,Z 382.795,A -85,B 0,C 180,E1 -374.721,E2 -374.721} C_VEL
LIN {X 0,Y 608.458,Z 375.576,A -85,B 0,C 180,E1 -377.476,E2 -377.476} C_VEL
LIN {X 0,Y 608.443,Z 368.356,A -85,B 0,C 180,E1 -380.275,E2 -380.275} C_VEL
LIN {X 0,Y 608.446,Z 361.136,A -85,B 0,C 180,E1 -383.124,E2 -383.124} C_VEL
LIN {X 0,Y 608.465,Z 354.69,A -85,B 0,C 180,E1 -385.719,E2 -385.719} C_VEL
LIN {X 0,Y 608.481,Z 347.629,A -85,B 0,C 180,E1 -388.621,E2 -388.621} C_VEL
LIN {X 0,Y 608.472,Z 344.693,A -85,B 0,C 180,E1 -389.906,E2 -389.906} C_VEL
LIN {X 0,Y 608.457,Z 344.696,A -85,B 0,C 180,E1 -392.88,E2 -392.88} C_VEL
LIN {X 0,Y 608.444,Z 344.696,A -85,B 0,C 180,E1 -395.278,E2 -395.278} C_VEL
LIN {X 0,Y 608.469,Z 344.694,A -85,B 0,C 180,E1 -397.746,E2 -397.746} C_VEL
LIN {X 0,Y 608.456,Z 344.696,A -85,B 0,C 180,E1 -400.329,E2 -400.329} C_VEL
LIN {X 0,Y 608.456,Z 344.696,A -85,B 0,C 180,E1 -402.96,E2 -402.96} C_VEL
LIN {X 0,Y 608.463,Z 344.694,A -85,B 0,C 180,E1 -405.736,E2 -405.736} C_VEL
LIN {X 0,Y 608.468,Z 344.695,A -85,B 0,C 180,E1 -408.657,E2 -408.657} C_VEL
LIN {X 0,Y 608.463,Z 344.696,A -85,B 0,C 180,E1 -411.76,E2 -411.76} C_VEL
LIN {X 0,Y 608.449,Z 344.697,A -85,B 0,C 180,E1 -413.955,E2 -413.955} C_VEL
LIN {X 0,Y 608.47,Z 344.693,A -85,B 0,C 180,E1 -416.329,E2 -416.329} C_VEL
LIN {X 0,Y 608.45,Z 344.697,A -85,B 0,C 180,E1 -418.732,E2 -418.732} C_VEL
LIN {X 0,Y 608.48,Z 344.693,A -85,B 0,C 180,E1 -421.379,E2 -421.379} C_VEL
LIN {X 0,Y 608.482,Z 344.705,A -85,B 0,C 180,E1 -422.39,E2 -422.39} C_VEL
LIN {X 0,Y 608.617,Z 357.706,A -85,B 0,C 180,E1 -424.48,E2 -424.48} C_VEL
LIN {X 0,Y 608.571,Z 375.514,A -85,B 0,C 180,E1 -427.276,E2 -427.276} C_VEL
LIN {X 0,Y 608.516,Z 393.746,A -85,B 0,C 180,E1 -430.08,E2 -430.08} C_VEL
LIN {X 0,Y 608.5,Z 411.055,A -85,B 0,C 180,E1 -432.698,E2 -432.698} C_VEL
LIN {X 0,Y 608.471,Z 429.517,A -85,B 0,C 180,E1 -435.45,E2 -435.45} C_VEL
LIN {X 0,Y 608.486,Z 447.98,A -85,B 0,C 180,E1 -438.17,E2 -438.17} C_VEL
LIN {X 0,Y 608.545,Z 463.26,A -85,B 0,C 180,E1 -438.445,E2 -438.445} C_VEL
LIN {X 0,Y 608.523,Z 475.883,A -85,B 0,C 180,E1 -438.808,E2 -438.808} C_VEL
LIN {X 0,Y 608.519,Z 487.579,A -85,B 0,C 180,E1 -439.275,E2 -439.275} C_VEL
LIN {X 0,Y 608.492,Z 498.753,A -85,B 0,C 180,E1 -439.855,E2 -439.855} C_VEL
LIN {X 0,Y 608.504,Z 510.25,A -85,B 0,C 180,E1 -440.611,E2 -440.611} C_VEL
LIN {X 0,Y 608.472,Z 519.534,A -85,B 0,C 180,E1 -441.364,E2 -441.364} C_VEL
LIN {X 0,Y 608.456,Z 527.988,A -85,B 0,C 180,E1 -442.2,E2 -442.2} C_VEL
LIN {X 0,Y 608.462,Z 536.234,A -85,B 0,C 180,E1 -443.201,E2 -443.201} C_VEL
LIN {X 0,Y 608.437,Z 542.876,A -85,B 0,C 180,E1 -444.199,E2 -444.199} C_VEL
LIN {X 0,Y 608.432,Z 548.949,A -85,B 0,C 180,E1 -445.362,E2 -445.362} C_VEL
LIN {X 0,Y 608.449,Z 552.896,A -85,B 0,C 180,E1 -446.357,E2 -446.357} C_VEL
LIN {X 0,Y 608.425,Z 555.809,A -85,B 0,C 180,E1 -447.352,E2 -447.352} C_VEL
LIN {X 0,Y 608.444,Z 557.201,A -85,B 0,C 180,E1 -448.014,E2 -448.014} C_VEL
LIN {X 0,Y 608.438,Z 558.783,A -85,B 0,C 180,E1 -449.338,E2 -449.338} C_VEL
LIN {X 0,Y 608.434,Z 559,A -85,B 0,C 180,E1 -450,E2 -450} C_VEL
LIN {X 0,Y 608.448,Z 558.184,A -85,B 0,C 180,E1 -451.324,E2 -451.324} C_VEL
LIN {X 0,Y 608.444,Z 557.202,A -85,B 0,C 180,E1 -451.986,E2 -451.986} C_VEL
LIN {X 0,Y 608.425,Z 555.809,A -85,B 0,C 180,E1 -452.648,E2 -452.648} C_VEL
LIN {X 0,Y 608.449,Z 552.897,A -85,B 0,C 180,E1 -453.642,E2 -453.642} C_VEL
LIN {X 0,Y 608.432,Z 548.951,A -85,B 0,C 180,E1 -454.638,E2 -454.638} C_VEL
LIN {X 0,Y 608.437,Z 542.877,A -85,B 0,C 180,E1 -455.801,E2 -455.801} C_VEL
LIN {X 0,Y 608.462,Z 536.236,A -85,B 0,C 180,E1 -456.799,E2 -456.799} C_VEL
LIN {X 0,Y 608.456,Z 527.99,A -85,B 0,C 180,E1 -457.8,E2 -457.8} C_VEL
LIN {X 0,Y 608.472,Z 519.537,A -85,B 0,C 180,E1 -458.636,E2 -458.636} C_VEL
LIN {X 0,Y 608.481,Z 509.092,A -85,B 0,C 180,E1 -459.473,E2 -459.473} C_VEL
LIN {X 0,Y 608.492,Z 498.757,A -85,B 0,C 180,E1 -460.145,E2 -460.145} C_VEL
LIN {X 0,Y 608.521,Z 487.263,A -85,B 0,C 180,E1 -460.74,E2 -460.74} C_VEL
LIN {X 0,Y 608.529,Z 474.887,A -85,B 0,C 180,E1 -461.225,E2 -461.225} C_VEL
LIN {X 0,Y 608.546,Z 461.443,A -85,B 0,C 180,E1 -461.597,E2 -461.597} C_VEL
LIN {X 0,Y 608.486,Z 447.982,A -85,B 0,C 180,E1 -461.83,E2 -461.83} C_VEL
LIN {X 0,Y 608.489,Z 428.365,A -85,B 0,C 180,E1 -464.72,E2 -464.72} C_VEL
LIN {X 0,Y 608.502,Z 409.902,A -85,B 0,C 180,E1 -467.475,E2 -467.475} C_VEL
LIN {X 0,Y 608.531,Z 392.594,A -85,B 0,C 180,E1 -470.095,E2 -470.095} C_VEL
LIN {X 0,Y 608.571,Z 374.132,A -85,B 0,C 180,E1 -472.939,E2 -472.939} C_VEL
LIN {X 0,Y 608.614,Z 356.269,A -85,B 0,C 180,E1 -475.748,E2 -475.748} C_VEL
LIN {X 0,Y 608.479,Z 344.706,A -85,B 0,C 180,E1 -477.61,E2 -477.61} C_VEL
LIN {X 0,Y 608.473,Z 344.69,A -85,B 0,C 180,E1 -480.545,E2 -480.545} C_VEL
LIN {X 0,Y 608.461,Z 344.69,A -85,B 0,C 180,E1 -482.879,E2 -482.879} C_VEL
LIN {X 0,Y 608.444,Z 344.697,A -85,B 0,C 180,E1 -485.278,E2 -485.278} C_VEL
LIN {X 0,Y 608.466,Z 344.689,A -85,B 0,C 180,E1 -487.746,E2 -487.746} C_VEL
LIN {X 0,Y 608.452,Z 344.696,A -85,B 0,C 180,E1 -490.329,E2 -490.329} C_VEL
LIN {X 0,Y 608.452,Z 344.692,A -85,B 0,C 180,E1 -492.96,E2 -492.96} C_VEL
LIN {X 0,Y 608.45,Z 344.692,A -85,B 0,C 180,E1 -495.737,E2 -495.737} C_VEL
LIN {X 0,Y 608.461,Z 344.69,A -85,B 0,C 180,E1 -497.938,E2 -497.938} C_VEL
LIN {X 0,Y 608.476,Z 344.689,A -85,B 0,C 180,E1 -500.702,E2 -500.702} C_VEL
LIN {X 0,Y 608.459,Z 344.692,A -85,B 0,C 180,E1 -503.085,E2 -503.085} C_VEL
LIN {X 0,Y 608.475,Z 344.691,A -85,B 0,C 180,E1 -505.531,E2 -505.531} C_VEL
LIN {X 0,Y 608.464,Z 344.69,A -85,B 0,C 180,E1 -507.905,E2 -507.905} C_VEL
LIN {X 0,Y 608.482,Z 344.694,A -85,B 0,C 180,E1 -510.221,E2 -510.221} C_VEL
LIN {X 0,Y 608.459,Z 344.693,A -85,B 0,C 180,E1 -513.226,E2 -513.226} C_VEL
LIN {X 0,Y 608.466,Z 344.689,A -85,B 0,C 180,E1 -516.155,E2 -516.155} C_VEL
LIN {X 0,Y 608.456,Z 344.691,A -85,B 0,C 180,E1 -519.018,E2 -519.018} C_VEL
LIN {X 0,Y 608.444,Z 344.698,A -85,B 0,C 180,E1 -521.828,E2 -521.828} C_VEL
LIN {X 0,Y 608.471,Z 344.689,A -85,B 0,C 180,E1 -524.594,E2 -524.594} C_VEL
LIN {X 0,Y 608.479,Z 344.689,A -85,B 0,C 180,E1 -527.323,E2 -527.323} C_VEL
LIN {X 0,Y 608.464,Z 344.694,A -85,B 0,C 180,E1 -530.023,E2 -530.023} C_VEL
LIN {X 0,Y 608.463,Z 344.689,A -85,B 0,C 180,E1 -532.701,E2 -532.701} C_VEL
LIN {X 0,Y 608.463,Z 344.695,A -85,B 0,C 180,E1 -535.362,E2 -535.362} C_VEL
LIN {X 0,Y 608.448,Z 344.692,A -85,B 0,C 180,E1 -538.014,E2 -538.014} C_VEL
LIN {X 0,Y 608.479,Z 344.689,A -85,B 0,C 180,E1 -540.662,E2 -540.662} C_VEL
LIN {X 0,Y 608.478,Z 344.691,A -85,B 0,C 180,E1 -543.311,E2 -543.311} C_VEL
LIN {X 0,Y 608.453,Z 344.691,A -85,B 0,C 180,E1 -545.967,E2 -545.967} C_VEL
LIN {X 0,Y 608.465,Z 344.696,A -85,B 0,C 180,E1 -548.636,E2 -548.636} C_VEL
LIN {X 0,Y 608.461,Z 344.689,A -85,B 0,C 180,E1 -549.459,E2 -549.459} C_VEL
LIN {X 0,Y 607.778,Z 344.78,A -85,B 0,C 180,E1 -550.011,E2 -550.011} C_VEL
LIN {X 0,Y 604.925,Z 345.135,A -85,B 0,C 180,E1 -550.908,E2 -550.908} C_VEL
LIN {X 0,Y 602.525,Z 345.435,A -85,B 0,C 180,E1 -551.63,E2 -551.63} C_VEL
LIN {X 0,Y 601.496,Z 345.562,A -85,B 0,C 180,E1 -552.186,E2 -552.186} C_VEL
LIN {X 0,Y 601.412,Z 345.569,A -85,B 0,C 180,E1 -552.375,E2 -552.375} C_VEL
LIN {X 0,Y 601.428,Z 345.568,A -85,B 0,C 180,E1 -554.897,E2 -554.897} C_VEL
LIN {X 0,Y 601.433,Z 345.572,A -85,B 0,C 180,E1 -556.986,E2 -556.986} C_VEL
LIN {X 0,Y 601.409,Z 345.57,A -85,B 0,C 180,E1 -559.809,E2 -559.809} C_VEL
LIN {X 0,Y 601.414,Z 345.568,A -85,B 0,C 180,E1 -562.683,E2 -562.683} C_VEL
LIN {X 0,Y 601.405,Z 345.57,A -85,B 0,C 180,E1 -564.879,E2 -564.879} C_VEL
LIN {X 0,Y 601.42,Z 345.569,A -85,B 0,C 180,E1 -567.363,E2 -567.363} C_VEL
LIN {X 0,Y 601.431,Z 345.571,A -85,B 0,C 180,E1 -570.164,E2 -570.164} C_VEL
LIN {X 0,Y 601.418,Z 345.567,A -85,B 0,C 180,E1 -572.715,E2 -572.715} C_VEL
LIN {X 0,Y 601.413,Z 345.572,A -85,B 0,C 180,E1 -575.114,E2 -575.114} C_VEL
LIN {X 0,Y 601.436,Z 345.566,A -85,B 0,C 180,E1 -577.419,E2 -577.419} C_VEL
LIN {X 0,Y 601.413,Z 345.57,A -85,B 0,C 180,E1 -579.995,E2 -579.995} C_VEL
LIN {X 0,Y 601.412,Z 345.568,A -85,B 0,C 180,E1 -582.67,E2 -582.67} C_VEL
LIN {X 0,Y 601.428,Z 345.571,A -85,B 0,C 180,E1 -585.482,E2 -585.482} C_VEL
LIN {X 0,Y 601.425,Z 345.57,A -85,B 0,C 180,E1 -588.407,E2 -588.407} C_VEL
LIN {X 0,Y 601.435,Z 345.566,A -85,B 0,C 180,E1 -591.529,E2 -591.529} C_VEL
LIN {X 0,Y 601.389,Z 345.571,A -85,B 0,C 180,E1 -594.246,E2 -594.246} C_VEL
LIN {X 0,Y 601.431,Z 345.568,A -85,B 0,C 180,E1 -596.687,E2 -596.687} C_VEL
LIN {X 0,Y 601.414,Z 345.569,A -85,B 0,C 180,E1 -599.058,E2 -599.058} C_VEL
LIN {X 0,Y 601.433,Z 345.565,A -85,B 0,C 180,E1 -601.373,E2 -601.373} C_VEL
LIN {X 0,Y 601.419,Z 345.569,A -85,B 0,C 180,E1 -604.132,E2 -604.132} C_VEL
LIN {X 0,Y 601.422,Z 345.568,A -85,B 0,C 180,E1 -606.59,E2 -606.59} C_VEL
LIN {X 0,Y 601.431,Z 345.565,A -85,B 0,C 180,E1 -609.478,E2 -609.478} C_VEL
LIN {X 0,Y 601.399,Z 345.573,A -85,B 0,C 180,E1 -612.312,E2 -612.312} C_VEL
LIN {X 0,Y 601.414,Z 345.568,A -85,B 0,C 180,E1 -614.409,E2 -614.409} C_VEL
LIN {X 0,Y 601.42,Z 345.572,A -85,B 0,C 180,E1 -617.172,E2 -617.172} C_VEL
LIN {X 0,Y 601.44,Z 345.565,A -85,B 0,C 180,E1 -619.905,E2 -619.905} C_VEL
LIN {X 0,Y 601.441,Z 345.565,A -85,B 0,C 180,E1 -622.615,E2 -622.615} C_VEL
LIN {X 0,Y 601.431,Z 345.572,A -85,B 0,C 180,E1 -625.308,E2 -625.308} C_VEL
LIN {X 0,Y 601.437,Z 345.565,A -85,B 0,C 180,E1 -627.991,E2 -627.991} C_VEL
LIN {X 0,Y 601.452,Z 345.566,A -85,B 0,C 180,E1 -630.67,E2 -630.67} C_VEL
LIN {X 0,Y 601.427,Z 345.568,A -85,B 0,C 180,E1 -633.35,E2 -633.35} C_VEL
LIN {X 0,Y 601.44,Z 345.565,A -85,B 0,C 180,E1 -636.037,E2 -636.037} C_VEL
LIN {X 0,Y 601.416,Z 345.575,A -85,B 0,C 180,E1 -638.738,E2 -638.738} C_VEL
LIN {X 0,Y 601.426,Z 345.566,A -85,B 0,C 180,E1 -641.458,E2 -641.458} C_VEL
LIN {X 0,Y 601.423,Z 345.568,A -85,B 0,C 180,E1 -644.206,E2 -644.206} C_VEL
LIN {X 0,Y 601.436,Z 345.571,A -85,B 0,C 180,E1 -646.986,E2 -646.986} C_VEL
LIN {X 0,Y 601.407,Z 345.569,A -85,B 0,C 180,E1 -649.81,E2 -649.81} C_VEL
LIN {X 0,Y 601.42,Z 345.568,A -85,B 0,C 180,E1 -652.606,E2 -652.606} C_VEL
LIN {X 0,Y 601.403,Z 345.569,A -85,B 0,C 180,E1 -654.879,E2 -654.879} C_VEL
LIN {X 0,Y 601.421,Z 345.57,A -85,B 0,C 180,E1 -657.363,E2 -657.363} C_VEL
LIN {X 0,Y 601.431,Z 345.569,A -85,B 0,C 180,E1 -660.164,E2 -660.164} C_VEL
LIN {X 0,Y 601.428,Z 345.566,A -85,B 0,C 180,E1 -662.716,E2 -662.716} C_VEL
LIN {X 0,Y 601.394,Z 345.572,A -85,B 0,C 180,E1 -665.111,E2 -665.111} C_VEL
LIN {X 0,Y 601.439,Z 345.568,A -85,B 0,C 180,E1 -667.419,E2 -667.419} C_VEL
LIN {X 0,Y 601.405,Z 345.57,A -85,B 0,C 180,E1 -669.996,E2 -669.996} C_VEL
LIN {X 0,Y 601.416,Z 345.568,A -85,B 0,C 180,E1 -672.67,E2 -672.67} C_VEL
LIN {X 0,Y 601.429,Z 345.566,A -85,B 0,C 180,E1 -674.535,E2 -674.535} C_VEL
LIN {X 0,Y 601.41,Z 345.571,A -85,B 0,C 180,E1 -677.41,E2 -677.41} C_VEL
LIN {X 0,Y 601.445,Z 345.571,A -85,B 0,C 180,E1 -680.464,E2 -680.464} C_VEL
LIN {X 0,Y 601.416,Z 345.569,A -85,B 0,C 180,E1 -683.418,E2 -683.418} C_VEL
LIN {X 0,Y 601.437,Z 345.565,A -85,B 0,C 180,E1 -686.064,E2 -686.064} C_VEL
LIN {X 0,Y 601.426,Z 345.57,A -85,B 0,C 180,E1 -689.058,E2 -689.058} C_VEL
LIN {X 0,Y 601.436,Z 345.77,A -85,B 0,C 180,E1 -690.319,E2 -690.319} C_VEL
LIN {X 0,Y 601.405,Z 351.909,A -85,B 0,C 180,E1 -692.887,E2 -692.887} C_VEL
LIN {X 0,Y 601.404,Z 358.759,A -85,B 0,C 180,E1 -695.715,E2 -695.715} C_VEL
LIN {X 0,Y 601.361,Z 364.519,A -85,B 0,C 180,E1 -698.039,E2 -698.039} C_VEL
LIN {X 0,Y 601.374,Z 371.735,A -85,B 0,C 180,E1 -700.9,E2 -700.9} C_VEL
LIN {X 0,Y 601.356,Z 378.951,A -85,B 0,C 180,E1 -703.711,E2 -703.711} C_VEL
LIN {X 0,Y 601.345,Z 386.167,A -85,B 0,C 180,E1 -706.482,E2 -706.482} C_VEL
LIN {X 0,Y 601.346,Z 393.384,A -85,B 0,C 180,E1 -709.223,E2 -709.223} C_VEL
LIN {X 0,Y 601.324,Z 400.601,A -85,B 0,C 180,E1 -711.938,E2 -711.938} C_VEL
LIN {X 0,Y 601.345,Z 403.682,A -85,B 0,C 180,E1 -713.091,E2 -713.091} C_VEL
LIN {X 0,Y 601.432,Z 413.86,A -85,B 0,C 180,E1 -713.447,E2 -713.447} C_VEL
LIN {X 0,Y 601.387,Z 422.194,A -85,B 0,C 180,E1 -713.862,E2 -713.862} C_VEL
LIN {X 0,Y 601.381,Z 430.191,A -85,B 0,C 180,E1 -714.383,E2 -714.383} C_VEL
LIN {X 0,Y 601.388,Z 437.032,A -85,B 0,C 180,E1 -714.972,E2 -714.972} C_VEL
LIN {X 0,Y 601.362,Z 443.21,A -85,B 0,C 180,E1 -715.643,E2 -715.643} C_VEL
LIN {X 0,Y 601.374,Z 448.071,A -85,B 0,C 180,E1 -716.315,E2 -716.315} C_VEL
LIN {X 0,Y 601.379,Z 451.821,A -85,B 0,C 180,E1 -716.985,E2 -716.985} C_VEL
LIN {X 0,Y 601.343,Z 455.827,A -85,B 0,C 180,E1 -717.991,E2 -717.991} C_VEL
LIN {X 0,Y 601.349,Z 457.57,A -85,B 0,C 180,E1 -718.661,E2 -718.661} C_VEL
LIN {X 0,Y 601.34,Z 458.616,A -85,B 0,C 180,E1 -719.33,E2 -719.33} C_VEL
LIN {X 0,Y 601.335,Z 458.996,A -85,B 0,C 180,E1 -720,E2 -720} C_VEL
LIN {X 0,Y 601.339,Z 458.714,A -85,B 0,C 180,E1 -720.67,E2 -720.67} C_VEL
LIN {X 0,Y 601.349,Z 457.767,A -85,B 0,C 180,E1 -721.339,E2 -721.339} C_VEL
LIN {X 0,Y 601.342,Z 456.127,A -85,B 0,C 180,E1 -722.009,E2 -722.009} C_VEL
LIN {X 0,Y 601.332,Z 453.743,A -85,B 0,C 180,E1 -722.68,E2 -722.68} C_VEL
LIN {X 0,Y 601.375,Z 448.615,A -85,B 0,C 180,E1 -723.685,E2 -723.685} C_VEL
LIN {X 0,Y 601.378,Z 442.551,A -85,B 0,C 180,E1 -724.524,E2 -724.524} C_VEL
LIN {X 0,Y 601.352,Z 436.243,A -85,B 0,C 180,E1 -725.197,E2 -725.197} C_VEL
LIN {X 0,Y 601.391,Z 429.087,A -85,B 0,C 180,E1 -725.785,E2 -725.785} C_VEL
LIN {X 0,Y 601.403,Z 420.6,A -85,B 0,C 180,E1 -726.318,E2 -726.318} C_VEL
LIN {X 0,Y 601.426,Z 411.076,A -85,B 0,C 180,E1 -726.753,E2 -726.753} C_VEL
LIN {X 0,Y 601.334,Z 403.661,A -85,B 0,C 180,E1 -727.007,E2 -727.007} C_VEL
LIN {X 0,Y 601.33,Z 397.232,A -85,B 0,C 180,E1 -729.417,E2 -729.417} C_VEL
LIN {X 0,Y 601.343,Z 390.013,A -85,B 0,C 180,E1 -732.144,E2 -732.144} C_VEL
LIN {X 0,Y 601.361,Z 382.794,A -85,B 0,C 180,E1 -734.899,E2 -734.899} C_VEL
LIN {X 0,Y 601.378,Z 375.574,A -85,B 0,C 180,E1 -737.689,E2 -737.689} C_VEL
LIN {X 0,Y 601.367,Z 368.354,A -85,B 0,C 180,E1 -740.524,E2 -740.524} C_VEL
LIN {X 0,Y 601.381,Z 361.134,A -85,B 0,C 180,E1 -743.412,E2 -743.412} C_VEL
LIN {X 0,Y 601.396,Z 355.126,A -85,B 0,C 180,E1 -745.863,E2 -745.863} C_VEL
LIN {X 0,Y 601.438,Z 348.445,A -85,B 0,C 180,E1 -748.627,E2 -748.627} C_VEL
LIN {X 0,Y 601.437,Z 345.57,A -85,B 0,C 180,E1 -749.871,E2 -749.871} C_VEL
LIN {X 0,Y 601.423,Z 345.574,A -85,B 0,C 180,E1 -752.715,E2 -752.715} C_VEL
LIN {X 0,Y 601.404,Z 345.574,A -85,B 0,C 180,E1 -755.113,E2 -755.113} C_VEL
LIN {X 0,Y 601.437,Z 345.569,A -85,B 0,C 180,E1 -757.419,E2 -757.419} C_VEL
LIN {X 0,Y 601.416,Z 345.574,A -85,B 0,C 180,E1 -759.995,E2 -759.995} C_VEL
LIN {X 0,Y 601.415,Z 345.572,A -85,B 0,C 180,E1 -762.67,E2 -762.67} C_VEL
LIN {X 0,Y 601.43,Z 345.572,A -85,B 0,C 180,E1 -765.482,E2 -765.482} C_VEL
LIN {X 0,Y 601.43,Z 345.573,A -85,B 0,C 180,E1 -768.407,E2 -768.407} C_VEL
LIN {X 0,Y 601.406,Z 345.574,A -85,B 0,C 180,E1 -770.873,E2 -770.873} C_VEL
LIN {X 0,Y 601.402,Z 345.574,A -85,B 0,C 180,E1 -773.417,E2 -773.417} C_VEL
LIN {X 0,Y 601.437,Z 345.57,A -85,B 0,C 180,E1 -776.064,E2 -776.064} C_VEL
LIN {X 0,Y 601.424,Z 345.571,A -85,B 0,C 180,E1 -778.545,E2 -778.545} C_VEL
LIN {X 0,Y 601.44,Z 345.571,A -85,B 0,C 180,E1 -781.373,E2 -781.373} C_VEL
LIN {X 0,Y 601.44,Z 345.694,A -85,B 0,C 180,E1 -782.201,E2 -782.201} C_VEL
LIN {X 0,Y 601.773,Z 349.897,A -85,B 0,C 180,E1 -782.904,E2 -782.904} C_VEL
LIN {X 0,Y 601.665,Z 367.049,A -85,B 0,C 180,E1 -785.66,E2 -785.66} C_VEL
LIN {X 0,Y 601.598,Z 384.515,A -85,B 0,C 180,E1 -788.408,E2 -788.408} C_VEL
LIN {X 0,Y 601.529,Z 402.274,A -85,B 0,C 180,E1 -791.151,E2 -791.151} C_VEL
LIN {X 0,Y 601.492,Z 421.44,A -85,B 0,C 180,E1 -794.063,E2 -794.063} C_VEL
LIN {X 0,Y 601.437,Z 441.056,A -85,B 0,C 180,E1 -797,E2 -797} C_VEL
LIN {X 0,Y 601.443,Z 448.19,A -85,B 0,C 180,E1 -798.04,E2 -798.04} C_VEL
LIN {X 0,Y 601.583,Z 461.432,A -85,B 0,C 180,E1 -798.267,E2 -798.267} C_VEL
LIN {X 0,Y 601.556,Z 474.218,A -85,B 0,C 180,E1 -798.621,E2 -798.621} C_VEL
LIN {X 0,Y 601.548,Z 485.843,A -85,B 0,C 180,E1 -799.072,E2 -799.072} C_VEL
LIN {X 0,Y 601.483,Z 497.324,A -85,B 0,C 180,E1 -799.651,E2 -799.651} C_VEL
LIN {X 0,Y 601.47,Z 507.929,A -85,B 0,C 180,E1 -800.33,E2 -800.33} C_VEL
LIN {X 0,Y 601.435,Z 517.597,A -85,B 0,C 180,E1 -801.093,E2 -801.093} C_VEL
LIN {X 0,Y 601.407,Z 526.412,A -85,B 0,C 180,E1 -801.939,E2 -801.939} C_VEL
LIN {X 0,Y 601.388,Z 533.689,A -85,B 0,C 180,E1 -802.783,E2 -802.783} C_VEL
LIN {X 0,Y 601.375,Z 540.773,A -85,B 0,C 180,E1 -803.782,E2 -803.782} C_VEL
LIN {X 0,Y 601.373,Z 545.679,A -85,B 0,C 180,E1 -804.635,E2 -804.635} C_VEL
LIN {X 0,Y 601.353,Z 550.37,A -85,B 0,C 180,E1 -805.643,E2 -805.643} C_VEL
LIN {X 0,Y 601.344,Z 553.956,A -85,B 0,C 180,E1 -806.65,E2 -806.65} C_VEL
LIN {X 0,Y 601.325,Z 555.809,A -85,B 0,C 180,E1 -807.32,E2 -807.32} C_VEL
LIN {X 0,Y 601.343,Z 557.201,A -85,B 0,C 180,E1 -807.991,E2 -807.991} C_VEL
LIN {X 0,Y 601.339,Z 558.784,A -85,B 0,C 180,E1 -809.33,E2 -809.33} C_VEL
LIN {X 0,Y 601.335,Z 559,A -85,B 0,C 180,E1 -810,E2 -810} C_VEL
LIN {X 0,Y 601.348,Z 558.184,A -85,B 0,C 180,E1 -811.339,E2 -811.339} C_VEL
LIN {X 0,Y 601.343,Z 557.202,A -85,B 0,C 180,E1 -812.009,E2 -812.009} C_VEL
LIN {X 0,Y 601.325,Z 555.81,A -85,B 0,C 180,E1 -812.679,E2 -812.679} C_VEL
LIN {X 0,Y 601.367,Z 552.897,A -85,B 0,C 180,E1 -813.685,E2 -813.685} C_VEL
LIN {X 0,Y 601.336,Z 548.951,A -85,B 0,C 180,E1 -814.693,E2 -814.693} C_VEL
LIN {X 0,Y 601.372,Z 542.878,A -85,B 0,C 180,E1 -815.869,E2 -815.869} C_VEL
LIN {X 0,Y 601.382,Z 536.236,A -85,B 0,C 180,E1 -816.88,E2 -816.88} C_VEL
LIN {X 0,Y 601.4,Z 527.99,A -85,B 0,C 180,E1 -817.892,E2 -817.892} C_VEL
LIN {X 0,Y 601.436,Z 519.538,A -85,B 0,C 180,E1 -818.738,E2 -818.738} C_VEL
LIN {X 0,Y 601.451,Z 509.093,A -85,B 0,C 180,E1 -819.585,E2 -819.585} C_VEL
LIN {X 0,Y 601.471,Z 498.758,A -85,B 0,C 180,E1 -820.264,E2 -820.264} C_VEL
LIN {X 0,Y 601.537,Z 487.912,A -85,B 0,C 180,E1 -820.835,E2 -820.835} C_VEL
LIN {X 0,Y 601.552,Z 475.385,A -85,B 0,C 180,E1 -821.34,E2 -821.34} C_VEL
LIN {X 0,Y 601.577,Z 462.356,A -85,B 0,C 180,E1 -821.711,E2 -821.711} C_VEL
LIN {X 0,Y 601.589,Z 449.091,A -85,B 0,C 180,E1 -821.946,E2 -821.946} C_VEL
LIN {X 0,Y 601.424,Z 447.982,A -85,B 0,C 180,E1 -821.971,E2 -821.971} C_VEL
LIN {X 0,Y 601.478,Z 428.365,A -85,B 0,C 180,E1 -824.896,E2 -824.896} C_VEL
LIN {X 0,Y 601.511,Z 411.056,A -85,B 0,C 180,E1 -827.509,E2 -827.509} C_VEL
LIN {X 0,Y 601.583,Z 393.748,A -85,B 0,C 180,E1 -830.159,E2 -830.159} C_VEL
LIN {X 0,Y 601.635,Z 375.285,A -85,B 0,C 180,E1 -833.037,E2 -833.037} C_VEL
LIN {X 0,Y 601.733,Z 357.107,A -85,B 0,C 180,E1 -835.93,E2 -835.93} C_VEL
LIN {X 0,Y 601.703,Z 346.931,A -85,B 0,C 180,E1 -837.583,E2 -837.583} C_VEL
LIN {X 0,Y 601.418,Z 345.571,A -85,B 0,C 180,E1 -837.834,E2 -837.834} C_VEL
LIN {X 0,Y 601.431,Z 345.573,A -85,B 0,C 180,E1 -840.164,E2 -840.164} C_VEL
LIN {X 0,Y 601.427,Z 345.566,A -85,B 0,C 180,E1 -842.716,E2 -842.716} C_VEL
LIN {X 0,Y 601.4,Z 345.576,A -85,B 0,C 180,E1 -845.112,E2 -845.112} C_VEL
LIN {X 0,Y 601.436,Z 345.565,A -85,B 0,C 180,E1 -847.419,E2 -847.419} C_VEL
LIN {X 0,Y 601.403,Z 345.574,A -85,B 0,C 180,E1 -849.996,E2 -849.996} C_VEL
LIN {X 0,Y 601.415,Z 345.567,A -85,B 0,C 180,E1 -852.67,E2 -852.67} C_VEL
LIN {X 0,Y 601.428,Z 345.569,A -85,B 0,C 180,E1 -855.482,E2 -855.482} C_VEL
LIN {X 0,Y 601.426,Z 345.572,A -85,B 0,C 180,E1 -858.407,E2 -858.407} C_VEL
LIN {X 0,Y 601.437,Z 345.565,A -85,B 0,C 180,E1 -860.875,E2 -860.875} C_VEL
LIN {X 0,Y 601.447,Z 345.568,A -85,B 0,C 180,E1 -863.734,E2 -863.734} C_VEL
LIN {X 0,Y 601.426,Z 345.571,A -85,B 0,C 180,E1 -866.686,E2 -866.686} C_VEL
LIN {X 0,Y 601.432,Z 345.566,A -85,B 0,C 180,E1 -869.059,E2 -869.059} C_VEL
LIN {X 0,Y 601.429,Z 345.567,A -85,B 0,C 180,E1 -871.373,E2 -871.373} C_VEL
LIN {X 0,Y 601.407,Z 345.574,A -85,B 0,C 180,E1 -873.636,E2 -873.636} C_VEL
LIN {X 0,Y 601.461,Z 345.562,A -85,B 0,C 180,E1 -875.86,E2 -875.86} C_VEL
LIN {X 0,Y 601.411,Z 345.572,A -85,B 0,C 180,E1 -878.761,E2 -878.761} C_VEL
LIN {X 0,Y 601.417,Z 345.57,A -85,B 0,C 180,E1 -881.608,E2 -881.608} C_VEL
LIN {X 0,Y 601.441,Z 345.569,A -85,B 0,C 180,E1 -883.713,E2 -883.713} C_VEL
LIN {X 0,Y 601.423,Z 345.568,A -85,B 0,C 180,E1 -886.484,E2 -886.484} C_VEL
LIN {X 0,Y 601.416,Z 345.567,A -85,B 0,C 180,E1 -889.224,E2 -889.224} C_VEL
LIN {X 0,Y 601.44,Z 345.571,A -85,B 0,C 180,E1 -891.939,E2 -891.939} C_VEL
LIN {X 0,Y 601.428,Z 345.566,A -85,B 0,C 180,E1 -894.636,E2 -894.636} C_VEL
LIN {X 0,Y 601.449,Z 345.565,A -85,B 0,C 180,E1 -897.321,E2 -897.321} C_VEL
LIN {X 0,Y 601.448,Z 345.567,A -85,B 0,C 180,E1 -900,E2 -900} C_VEL
LIN {X 0,Y 601.444,Z 345.564,A -85,B 0,C 180,E1 -902.679,E2 -902.679} C_VEL
LIN {X 0,Y 601.435,Z 345.571,A -85,B 0,C 180,E1 -905.364,E2 -905.364} C_VEL
LIN {X 0,Y 601.439,Z 345.565,A -85,B 0,C 180,E1 -908.061,E2 -908.061} C_VEL
LIN {X 0,Y 601.425,Z 345.566,A -85,B 0,C 180,E1 -911.012,E2 -911.012} C_VEL
LIN {X 0,Y 601.412,Z 345.569,A -85,B 0,C 180,E1 -912.375,E2 -912.375} C_VEL
LIN {X 0,Y 600.745,Z 345.651,A -85,B 0,C 180,E1 -912.934,E2 -912.934} C_VEL
LIN {X 0,Y 597.894,Z 346.01,A -85,B 0,C 180,E1 -913.842,E2 -913.842} C_VEL
LIN {X 0,Y 595.484,Z 346.311,A -85,B 0,C 180,E1 -914.572,E2 -914.572} C_VEL
LIN {X 0,Y 594.446,Z 346.441,A -85,B 0,C 180,E1 -915.136,E2 -915.136} C_VEL
LIN {X 0,Y 594.359,Z 346.448,A -85,B 0,C 180,E1 -915.326,E2 -915.326} C_VEL
LIN {X 0,Y 594.356,Z 346.447,A -85,B 0,C 180,E1 -917.905,E2 -917.905} C_VEL
LIN {X 0,Y 594.404,Z 346.442,A -85,B 0,C 180,E1 -920.776,E2 -920.776} C_VEL
LIN {X 0,Y 594.392,Z 346.448,A -85,B 0,C 180,E1 -923.704,E2 -923.704} C_VEL
LIN {X 0,Y 594.387,Z 346.446,A -85,B 0,C 180,E1 -926.7,E2 -926.7} C_VEL
LIN {X 0,Y 594.383,Z 346.446,A -85,B 0,C 180,E1 -928.999,E2 -928.999} C_VEL
LIN {X 0,Y 594.378,Z 346.447,A -85,B 0,C 180,E1 -931.643,E2 -931.643} C_VEL
LIN {X 0,Y 594.396,Z 346.442,A -85,B 0,C 180,E1 -934.579,E2 -934.579} C_VEL
LIN {X 0,Y 594.39,Z 346.443,A -85,B 0,C 180,E1 -937.608,E2 -937.608} C_VEL
LIN {X 0,Y 594.372,Z 346.449,A -85,B 0,C 180,E1 -940.567,E2 -940.567} C_VEL
LIN {X 0,Y 594.368,Z 346.448,A -85,B 0,C 180,E1 -943.3,E2 -943.3} C_VEL
LIN {X 0,Y 594.385,Z 346.443,A -85,B 0,C 180,E1 -946.159,E2 -946.159} C_VEL
LIN {X 0,Y 594.378,Z 346.445,A -85,B 0,C 180,E1 -949.178,E2 -949.178} C_VEL
LIN {X 0,Y 594.39,Z 346.449,A -85,B 0,C 180,E1 -952.06,E2 -952.06} C_VEL
LIN {X 0,Y 594.356,Z 346.447,A -85,B 0,C 180,E1 -954.676,E2 -954.676} C_VEL
LIN {X 0,Y 594.383,Z 346.45,A -85,B 0,C 180,E1 -957.088,E2 -957.088} C_VEL
LIN {X 0,Y 594.387,Z 346.443,A -85,B 0,C 180,E1 -959.672,E2 -959.672} C_VEL
LIN {X 0,Y 594.377,Z 346.445,A -85,B 0,C 180,E1 -962.539,E2 -962.539} C_VEL
LIN {X 0,Y 594.379,Z 346.445,A -85,B 0,C 180,E1 -964.807,E2 -964.807} C_VEL
LIN {X 0,Y 594.369,Z 346.449,A -85,B 0,C 180,E1 -967.265,E2 -967.265} C_VEL
LIN {X 0,Y 594.373,Z 346.446,A -85,B 0,C 180,E1 -969.946,E2 -969.946} C_VEL
LIN {X 0,Y 594.392,Z 346.442,A -85,B 0,C 180,E1 -972.807,E2 -972.807} C_VEL
LIN {X 0,Y 594.393,Z 346.444,A -85,B 0,C 180,E1 -975.826,E2 -975.826} C_VEL
LIN {X 0,Y 594.397,Z 346.445,A -85,B 0,C 180,E1 -978.404,E2 -978.404} C_VEL
LIN {X 0,Y 594.381,Z 346.443,A -85,B 0,C 180,E1 -981.158,E2 -981.158} C_VEL
LIN {X 0,Y 594.39,Z 346.447,A -85,B 0,C 180,E1 -983.891,E2 -983.891} C_VEL
LIN {X 0,Y 594.379,Z 346.446,A -85,B 0,C 180,E1 -986.611,E2 -986.611} C_VEL
LIN {X 0,Y 594.42,Z 346.439,A -85,B 0,C 180,E1 -989.323,E2 -989.323} C_VEL
LIN {X 0,Y 594.406,Z 346.447,A -85,B 0,C 180,E1 -992.033,E2 -992.033} C_VEL
LIN {X 0,Y 594.389,Z 346.443,A -85,B 0,C 180,E1 -994.748,E2 -994.748} C_VEL
LIN {X 0,Y 594.399,Z 346.444,A -85,B 0,C 180,E1 -997.473,E2 -997.473} C_VEL
LIN {X 0,Y 594.403,Z 346.445,A -85,B 0,C 180,E1 -1000.216,E2 -1000.216} C_VEL
LIN {X 0,Y 594.365,Z 346.445,A -85,B 0,C 180,E1 -1002.983,E2 -1002.983} C_VEL
LIN {X 0,Y 594.374,Z 346.447,A -85,B 0,C 180,E1 -1005.078,E2 -1005.078} C_VEL
LIN {X 0,Y 594.394,Z 346.448,A -85,B 0,C 180,E1 -1007.193,E2 -1007.193} C_VEL
LIN {X 0,Y 594.378,Z 346.446,A -85,B 0,C 180,E1 -1010.054,E2 -1010.054} C_VEL
LIN {X 0,Y 594.367,Z 346.445,A -85,B 0,C 180,E1 -1012.967,E2 -1012.967} C_VEL
LIN {X 0,Y 594.379,Z 346.447,A -85,B 0,C 180,E1 -1015.193,E2 -1015.193} C_VEL
LIN {X 0,Y 594.39,Z 346.444,A -85,B 0,C 180,E1 -1017.527,E2 -1017.527} C_VEL
LIN {X 0,Y 594.388,Z 346.448,A -85,B 0,C 180,E1 -1020.328,E2 -1020.328} C_VEL
LIN {X 0,Y 594.384,Z 346.443,A -85,B 0,C 180,E1 -1022.95,E2 -1022.95} C_VEL
LIN {X 0,Y 594.352,Z 346.454,A -85,B 0,C 180,E1 -1025.409,E2 -1025.409} C_VEL
LIN {X 0,Y 594.388,Z 346.443,A -85,B 0,C 180,E1 -1027.941,E2 -1027.941} C_VEL
LIN {X 0,Y 594.381,Z 346.446,A -85,B 0,C 180,E1 -1030.822,E2 -1030.822} C_VEL
LIN {X 0,Y 594.387,Z 346.45,A -85,B 0,C 180,E1 -1033.841,E2 -1033.841} C_VEL
LIN {X 0,Y 594.369,Z 346.447,A -85,B 0,C 180,E1 -1036.7,E2 -1036.7} C_VEL
LIN {X 0,Y 594.369,Z 346.445,A -85,B 0,C 180,E1 -1039.433,E2 -1039.433} C_VEL
LIN {X 0,Y 594.392,Z 346.446,A -85,B 0,C 180,E1 -1042.392,E2 -1042.392} C_VEL
LIN {X 0,Y 594.361,Z 346.446,A -85,B 0,C 180,E1 -1044.676,E2 -1044.676} C_VEL
LIN {X 0,Y 594.379,Z 346.45,A -85,B 0,C 180,E1 -1047.089,E2 -1047.089} C_VEL
LIN {X 0,Y 594.391,Z 346.443,A -85,B 0,C 180,E1 -1049.672,E2 -1049.672} C_VEL
LIN {X 0,Y 594.413,Z 346.661,A -85,B 0,C 180,E1 -1050.323,E2 -1050.323} C_VEL
LIN {X 0,Y 594.365,Z 353.78,A -85,B 0,C 180,E1 -1053.299,E2 -1053.299} C_VEL
LIN {X 0,Y 594.34,Z 359.172,A -85,B 0,C 180,E1 -1055.577,E2 -1055.577} C_VEL
LIN {X 0,Y 594.285,Z 366.325,A -85,B 0,C 180,E1 -1058.494,E2 -1058.494} C_VEL
LIN {X 0,Y 594.288,Z 373.54,A -85,B 0,C 180,E1 -1061.379,E2 -1061.379} C_VEL
LIN {X 0,Y 594.276,Z 380.757,A -85,B 0,C 180,E1 -1064.217,E2 -1064.217} C_VEL
LIN {X 0,Y 594.26,Z 386.169,A -85,B 0,C 180,E1 -1066.318,E2 -1066.318} C_VEL
LIN {X 0,Y 594.243,Z 393.385,A -85,B 0,C 180,E1 -1069.092,E2 -1069.092} C_VEL
LIN {X 0,Y 594.251,Z 400.602,A -85,B 0,C 180,E1 -1071.841,E2 -1071.841} C_VEL
LIN {X 0,Y 594.251,Z 403.703,A -85,B 0,C 180,E1 -1073.016,E2 -1073.016} C_VEL
LIN {X 0,Y 594.392,Z 414.145,A -85,B 0,C 180,E1 -1073.382,E2 -1073.382} C_VEL
LIN {X 0,Y 594.341,Z 422.404,A -85,B 0,C 180,E1 -1073.8,E2 -1073.8} C_VEL
LIN {X 0,Y 594.311,Z 430.198,A -85,B 0,C 180,E1 -1074.316,E2 -1074.316} C_VEL
LIN {X 0,Y 594.323,Z 437.038,A -85,B 0,C 180,E1 -1074.912,E2 -1074.912} C_VEL
LIN {X 0,Y 594.286,Z 443.214,A -85,B 0,C 180,E1 -1075.591,E2 -1075.591} C_VEL
LIN {X 0,Y 594.3,Z 448.074,A -85,B 0,C 180,E1 -1076.271,E2 -1076.271} C_VEL
LIN {X 0,Y 594.278,Z 451.823,A -85,B 0,C 180,E1 -1076.949,E2 -1076.949} C_VEL
LIN {X 0,Y 594.243,Z 455.829,A -85,B 0,C 180,E1 -1077.967,E2 -1077.967} C_VEL
LIN {X 0,Y 594.249,Z 457.572,A -85,B 0,C 180,E1 -1078.645,E2 -1078.645} C_VEL
LIN {X 0,Y 594.24,Z 458.617,A -85,B 0,C 180,E1 -1079.322,E2 -1079.322} C_VEL
LIN {X 0,Y 594.236,Z 458.996,A -85,B 0,C 180,E1 -1080,E2 -1080} C_VEL
LIN {X 0,Y 594.24,Z 458.713,A -85,B 0,C 180,E1 -1080.678,E2 -1080.678} C_VEL
LIN {X 0,Y 594.248,Z 457.766,A -85,B 0,C 180,E1 -1081.355,E2 -1081.355} C_VEL
LIN {X 0,Y 594.242,Z 456.125,A -85,B 0,C 180,E1 -1082.033,E2 -1082.033} C_VEL
LIN {X 0,Y 594.237,Z 453.741,A -85,B 0,C 180,E1 -1082.712,E2 -1082.712} C_VEL
LIN {X 0,Y 594.3,Z 448.612,A -85,B 0,C 180,E1 -1083.729,E2 -1083.729} C_VEL
LIN {X 0,Y 594.31,Z 442.546,A -85,B 0,C 180,E1 -1084.578,E2 -1084.578} C_VEL
LIN {X 0,Y 594.271,Z 436.237,A -85,B 0,C 180,E1 -1085.259,E2 -1085.259} C_VEL
LIN {X 0,Y 594.315,Z 429.081,A -85,B 0,C 180,E1 -1085.854,E2 -1085.854} C_VEL
LIN {X 0,Y 594.339,Z 421.348,A -85,B 0,C 180,E1 -1086.35,E2 -1086.35} C_VEL
LIN {X 0,Y 594.391,Z 412.233,A -85,B 0,C 180,E1 -1086.79,E2 -1086.79} C_VEL
LIN {X 0,Y 594.245,Z 403.659,A -85,B 0,C 180,E1 -1087.091,E2 -1087.091} C_VEL
LIN {X 0,Y 594.249,Z 397.23,A -85,B 0,C 180,E1 -1089.531,E2 -1089.531} C_VEL
LIN {X 0,Y 594.244,Z 390.011,A -85,B 0,C 180,E1 -1092.291,E2 -1092.291} C_VEL
LIN {X 0,Y 594.278,Z 382.792,A -85,B 0,C 180,E1 -1095.08,E2 -1095.08} C_VEL
LIN {X 0,Y 594.298,Z 377.378,A -85,B 0,C 180,E1 -1097.196,E2 -1097.196} C_VEL
LIN {X 0,Y 594.294,Z 370.158,A -85,B 0,C 180,E1 -1100.057,E2 -1100.057} C_VEL
LIN {X 0,Y 594.302,Z 362.938,A -85,B 0,C 180,E1 -1102.97,E2 -1102.97} C_VEL
LIN {X 0,Y 594.337,Z 357.523,A -85,B 0,C 180,E1 -1105.195,E2 -1105.195} C_VEL
LIN {X 0,Y 594.372,Z 352.064,A -85,B 0,C 180,E1 -1107.523,E2 -1107.523} C_VEL
LIN {X 0,Y 594.393,Z 346.448,A -85,B 0,C 180,E1 -1109.863,E2 -1109.863} C_VEL
LIN {X 0,Y 594.381,Z 346.45,A -85,B 0,C 180,E1 -1112.911,E2 -1112.911} C_VEL
LIN {X 0,Y 594.356,Z 346.452,A -85,B 0,C 180,E1 -1115.409,E2 -1115.409} C_VEL
LIN {X 0,Y 594.389,Z 346.45,A -85,B 0,C 180,E1 -1117.941,E2 -1117.941} C_VEL
LIN {X 0,Y 594.383,Z 346.448,A -85,B 0,C 180,E1 -1120.822,E2 -1120.822} C_VEL
LIN {X 0,Y 594.387,Z 346.448,A -85,B 0,C 180,E1 -1123.841,E2 -1123.841} C_VEL
LIN {X 0,Y 594.384,Z 346.448,A -85,B 0,C 180,E1 -1126.702,E2 -1126.702} C_VEL
LIN {X 0,Y 594.373,Z 346.451,A -85,B 0,C 180,E1 -1129.433,E2 -1129.433} C_VEL
LIN {X 0,Y 594.391,Z 346.448,A -85,B 0,C 180,E1 -1132.392,E2 -1132.392} C_VEL
LIN {X 0,Y 594.384,Z 346.448,A -85,B 0,C 180,E1 -1135.42,E2 -1135.42} C_VEL
LIN {X 0,Y 594.382,Z 346.449,A -85,B 0,C 180,E1 -1138.357,E2 -1138.357} C_VEL
LIN {X 0,Y 594.389,Z 346.45,A -85,B 0,C 180,E1 -1141.042,E2 -1141.042} C_VEL
LIN {X 0,Y 594.432,Z 346.599,A -85,B 0,C 180,E1 -1141.995,E2 -1141.995} C_VEL
LIN {X 0,Y 594.892,Z 349.897,A -85,B 0,C 180,E1 -1142.565,E2 -1142.565} C_VEL
LIN {X 0,Y 594.786,Z 366.283,A -85,B 0,C 180,E1 -1145.236,E2 -1145.236} C_VEL
LIN {X 0,Y 594.659,Z 384.515,A -85,B 0,C 180,E1 -1148.143,E2 -1148.143} C_VEL
LIN {X 0,Y 594.581,Z 402.157,A -85,B 0,C 180,E1 -1150.904,E2 -1150.904} C_VEL
LIN {X 0,Y 594.49,Z 421.44,A -85,B 0,C 180,E1 -1153.87,E2 -1153.87} C_VEL
LIN {X 0,Y 594.422,Z 439.902,A -85,B 0,C 180,E1 -1156.67,E2 -1156.67} C_VEL
LIN {X 0,Y 594.401,Z 448.19,A -85,B 0,C 180,E1 -1157.896,E2 -1157.896} C_VEL
LIN {X 0,Y 594.646,Z 454.938,A -85,B 0,C 180,E1 -1157.998,E2 -1157.998} C_VEL
LIN {X 0,Y 594.603,Z 468.212,A -85,B 0,C 180,E1 -1158.3,E2 -1158.3} C_VEL
LIN {X 0,Y 594.599,Z 480.415,A -85,B 0,C 180,E1 -1158.713,E2 -1158.713} C_VEL
LIN {X 0,Y 594.538,Z 492.63,A -85,B 0,C 180,E1 -1159.27,E2 -1159.27} C_VEL
LIN {X 0,Y 594.48,Z 504.197,A -85,B 0,C 180,E1 -1159.958,E2 -1159.958} C_VEL
LIN {X 0,Y 594.414,Z 514.594,A -85,B 0,C 180,E1 -1160.729,E2 -1160.729} C_VEL
LIN {X 0,Y 594.383,Z 523.11,A -85,B 0,C 180,E1 -1161.5,E2 -1161.5} C_VEL
LIN {X 0,Y 594.347,Z 530.959,A -85,B 0,C 180,E1 -1162.355,E2 -1162.355} C_VEL
LIN {X 0,Y 594.283,Z 538.812,A -85,B 0,C 180,E1 -1163.408,E2 -1163.408} C_VEL
LIN {X 0,Y 594.289,Z 545.68,A -85,B 0,C 180,E1 -1164.571,E2 -1164.571} C_VEL
LIN {X 0,Y 594.27,Z 550.371,A -85,B 0,C 180,E1 -1165.591,E2 -1165.591} C_VEL
LIN {X 0,Y 594.267,Z 553.956,A -85,B 0,C 180,E1 -1166.61,E2 -1166.61} C_VEL
LIN {X 0,Y 594.226,Z 555.808,A -85,B 0,C 180,E1 -1167.288,E2 -1167.288} C_VEL
LIN {X 0,Y 594.242,Z 557.201,A -85,B 0,C 180,E1 -1167.967,E2 -1167.967} C_VEL
LIN {X 0,Y 594.239,Z 558.784,A -85,B 0,C 180,E1 -1169.322,E2 -1169.322} C_VEL
LIN {X 0,Y 594.236,Z 559,A -85,B 0,C 180,E1 -1170,E2 -1170} C_VEL
LIN {X 0,Y 594.248,Z 558.185,A -85,B 0,C 180,E1 -1171.355,E2 -1171.355} C_VEL
LIN {X 0,Y 594.242,Z 557.202,A -85,B 0,C 180,E1 -1172.033,E2 -1172.033} C_VEL
LIN {X 0,Y 594.226,Z 555.81,A -85,B 0,C 180,E1 -1172.711,E2 -1172.711} C_VEL
LIN {X 0,Y 594.288,Z 552.897,A -85,B 0,C 180,E1 -1173.729,E2 -1173.729} C_VEL
LIN {X 0,Y 594.241,Z 548.95,A -85,B 0,C 180,E1 -1174.749,E2 -1174.749} C_VEL
LIN {X 0,Y 594.304,Z 542.878,A -85,B 0,C 180,E1 -1175.939,E2 -1175.939} C_VEL
LIN {X 0,Y 594.308,Z 536.237,A -85,B 0,C 180,E1 -1176.962,E2 -1176.962} C_VEL
LIN {X 0,Y 594.359,Z 527.991,A -85,B 0,C 180,E1 -1177.986,E2 -1177.986} C_VEL
LIN {X 0,Y 594.382,Z 519.538,A -85,B 0,C 180,E1 -1178.842,E2 -1178.842} C_VEL
LIN {X 0,Y 594.435,Z 509.094,A -85,B 0,C 180,E1 -1179.699,E2 -1179.699} C_VEL
LIN {X 0,Y 594.484,Z 498.76,A -85,B 0,C 180,E1 -1180.386,E2 -1180.386} C_VEL
LIN {X 0,Y 594.559,Z 487.706,A -85,B 0,C 180,E1 -1180.974,E2 -1180.974} C_VEL
LIN {X 0,Y 594.58,Z 475.707,A -85,B 0,C 180,E1 -1181.464,E2 -1181.464} C_VEL
LIN {X 0,Y 594.636,Z 462.355,A -85,B 0,C 180,E1 -1181.85,E2 -1181.85} C_VEL
LIN {X 0,Y 594.511,Z 449.091,A -85,B 0,C 180,E1 -1182.091,E2 -1182.091} C_VEL
LIN {X 0,Y 594.384,Z 447.982,A -85,B 0,C 180,E1 -1182.115,E2 -1182.115} C_VEL
LIN {X 0,Y 594.46,Z 428.365,A -85,B 0,C 180,E1 -1185.076,E2 -1185.076} C_VEL
LIN {X 0,Y 594.528,Z 411.056,A -85,B 0,C 180,E1 -1187.722,E2 -1187.722} C_VEL
LIN {X 0,Y 594.617,Z 393.748,A -85,B 0,C 180,E1 -1190.406,E2 -1190.406} C_VEL
LIN {X 0,Y 594.703,Z 375.285,A -85,B 0,C 180,E1 -1193.322,E2 -1193.322} C_VEL
LIN {X 0,Y 594.847,Z 357.96,A -85,B 0,C 180,E1 -1196.113,E2 -1196.113} C_VEL
LIN {X 0,Y 594.873,Z 348.81,A -85,B 0,C 180,E1 -1197.616,E2 -1197.616} C_VEL
LIN {X 0,Y 594.394,Z 346.447,A -85,B 0,C 180,E1 -1198.051,E2 -1198.051} C_VEL
LIN {X 0,Y 594.383,Z 346.446,A -85,B 0,C 180,E1 -1200.559,E2 -1200.559} C_VEL
LIN {X 0,Y 594.382,Z 346.445,A -85,B 0,C 180,E1 -1202.95,E2 -1202.95} C_VEL
LIN {X 0,Y 594.353,Z 346.451,A -85,B 0,C 180,E1 -1205.409,E2 -1205.409} C_VEL
LIN {X 0,Y 594.386,Z 346.444,A -85,B 0,C 180,E1 -1207.941,E2 -1207.941} C_VEL
LIN {X 0,Y 594.379,Z 346.444,A -85,B 0,C 180,E1 -1210.822,E2 -1210.822} C_VEL
LIN {X 0,Y 594.385,Z 346.446,A -85,B 0,C 180,E1 -1213.841,E2 -1213.841} C_VEL
LIN {X 0,Y 594.381,Z 346.449,A -85,B 0,C 180,E1 -1216.702,E2 -1216.702} C_VEL
LIN {X 0,Y 594.368,Z 346.445,A -85,B 0,C 180,E1 -1219.433,E2 -1219.433} C_VEL
LIN {X 0,Y 594.392,Z 346.443,A -85,B 0,C 180,E1 -1222.391,E2 -1222.391} C_VEL
LIN {X 0,Y 594.36,Z 346.447,A -85,B 0,C 180,E1 -1224.675,E2 -1224.675} C_VEL
LIN {X 0,Y 594.379,Z 346.448,A -85,B 0,C 180,E1 -1227.089,E2 -1227.089} C_VEL
LIN {X 0,Y 594.39,Z 346.443,A -85,B 0,C 180,E1 -1229.671,E2 -1229.671} C_VEL
LIN {X 0,Y 594.376,Z 346.444,A -85,B 0,C 180,E1 -1232.539,E2 -1232.539} C_VEL
LIN {X 0,Y 594.376,Z 346.446,A -85,B 0,C 180,E1 -1234.807,E2 -1234.807} C_VEL
LIN {X 0,Y 594.364,Z 346.448,A -85,B 0,C 180,E1 -1237.265,E2 -1237.265} C_VEL
LIN {X 0,Y 594.377,Z 346.448,A -85,B 0,C 180,E1 -1239.946,E2 -1239.946} C_VEL
LIN {X 0,Y 594.391,Z 346.442,A -85,B 0,C 180,E1 -1242.807,E2 -1242.807} C_VEL
LIN {X 0,Y 594.391,Z 346.443,A -85,B 0,C 180,E1 -1245.826,E2 -1245.826} C_VEL
LIN {X 0,Y 594.395,Z 346.447,A -85,B 0,C 180,E1 -1248.404,E2 -1248.404} C_VEL
LIN {X 0,Y 594.383,Z 346.443,A -85,B 0,C 180,E1 -1251.158,E2 -1251.158} C_VEL
LIN {X 0,Y 594.365,Z 346.448,A -85,B 0,C 180,E1 -1253.891,E2 -1253.891} C_VEL
LIN {X 0,Y 594.388,Z 346.446,A -85,B 0,C 180,E1 -1256.611,E2 -1256.611} C_VEL
LIN {X 0,Y 594.422,Z 346.439,A -85,B 0,C 180,E1 -1259.323,E2 -1259.323} C_VEL
LIN {X 0,Y 594.403,Z 346.447,A -85,B 0,C 180,E1 -1262.033,E2 -1262.033} C_VEL
LIN {X 0,Y 594.396,Z 346.443,A -85,B 0,C 180,E1 -1264.748,E2 -1264.748} C_VEL
LIN {X 0,Y 594.397,Z 346.442,A -85,B 0,C 180,E1 -1267.473,E2 -1267.473} C_VEL
LIN {X 0,Y 594.39,Z 346.449,A -85,B 0,C 180,E1 -1270.216,E2 -1270.216} C_VEL
LIN {X 0,Y 594.368,Z 346.446,A -85,B 0,C 180,E1 -1272.983,E2 -1272.983} C_VEL
LIN {X 0,Y 594.359,Z 346.448,A -85,B 0,C 180,E1 -1275.326,E2 -1275.326} C_VEL
LIN {X 0,Y 593.685,Z 346.532,A -85,B 0,C 180,E1 -1275.892,E2 -1275.892} C_VEL
LIN {X 0,Y 590.821,Z 346.892,A -85,B 0,C 180,E1 -1276.81,E2 -1276.81} C_VEL
LIN {X 0,Y 588.412,Z 347.19,A -85,B 0,C 180,E1 -1277.549,E2 -1277.549} C_VEL
LIN {X 0,Y 587.39,Z 347.316,A -85,B 0,C 180,E1 -1278.119,E2 -1278.119} C_VEL
LIN {X 0,Y 587.314,Z 347.325,A -85,B 0,C 180,E1 -1278.312,E2 -1278.312} C_VEL
LIN {X 0,Y 587.332,Z 347.322,A -85,B 0,C 180,E1 -1281.038,E2 -1281.038} C_VEL
LIN {X 0,Y 587.324,Z 347.325,A -85,B 0,C 180,E1 -1283.259,E2 -1283.259} C_VEL
LIN {X 0,Y 587.334,Z 347.325,A -85,B 0,C 180,E1 -1285.517,E2 -1285.517} C_VEL
LIN {X 0,Y 587.348,Z 347.319,A -85,B 0,C 180,E1 -1287.818,E2 -1287.818} C_VEL
LIN {X 0,Y 587.339,Z 347.325,A -85,B 0,C 180,E1 -1290.51,E2 -1290.51} C_VEL
LIN {X 0,Y 587.337,Z 347.325,A -85,B 0,C 180,E1 -1293.397,E2 -1293.397} C_VEL
LIN {X 0,Y 587.302,Z 347.326,A -85,B 0,C 180,E1 -1295.899,E2 -1295.899} C_VEL
LIN {X 0,Y 587.333,Z 347.326,A -85,B 0,C 180,E1 -1298.479,E2 -1298.479} C_VEL
LIN {X 0,Y 587.337,Z 347.321,A -85,B 0,C 180,E1 -1301.157,E2 -1301.157} C_VEL
LIN {X 0,Y 587.328,Z 347.324,A -85,B 0,C 180,E1 -1304.114,E2 -1304.114} C_VEL
LIN {X 0,Y 587.326,Z 347.33,A -85,B 0,C 180,E1 -1306.995,E2 -1306.995} C_VEL
LIN {X 0,Y 587.314,Z 347.324,A -85,B 0,C 180,E1 -1309.746,E2 -1309.746} C_VEL
LIN {X 0,Y 587.347,Z 347.322,A -85,B 0,C 180,E1 -1312.393,E2 -1312.393} C_VEL
LIN {X 0,Y 587.364,Z 347.319,A -85,B 0,C 180,E1 -1315.78,E2 -1315.78} C_VEL
LIN {X 0,Y 587.345,Z 347.322,A -85,B 0,C 180,E1 -1318.231,E2 -1318.231} C_VEL
LIN {X 0,Y 587.352,Z 347.32,A -85,B 0,C 180,E1 -1320.867,E2 -1320.867} C_VEL
LIN {X 0,Y 587.364,Z 347.323,A -85,B 0,C 180,E1 -1323.819,E2 -1323.819} C_VEL
LIN {X 0,Y 587.338,Z 347.321,A -85,B 0,C 180,E1 -1325.994,E2 -1325.994} C_VEL
LIN {X 0,Y 587.324,Z 347.324,A -85,B 0,C 180,E1 -1328.226,E2 -1328.226} C_VEL
LIN {X 0,Y 587.352,Z 347.319,A -85,B 0,C 180,E1 -1331.151,E2 -1331.151} C_VEL
LIN {X 0,Y 587.356,Z 347.321,A -85,B 0,C 180,E1 -1333.311,E2 -1333.311} C_VEL
LIN {X 0,Y 587.363,Z 347.318,A -85,B 0,C 180,E1 -1336.154,E2 -1336.154} C_VEL
LIN {X 0,Y 587.345,Z 347.324,A -85,B 0,C 180,E1 -1338.963,E2 -1338.963} C_VEL
LIN {X 0,Y 587.367,Z 347.32,A -85,B 0,C 180,E1 -1341.745,E2 -1341.745} C_VEL
LIN {X 0,Y 587.363,Z 347.318,A -85,B 0,C 180,E1 -1344.507,E2 -1344.507} C_VEL
LIN {X 0,Y 587.372,Z 347.321,A -85,B 0,C 180,E1 -1347.257,E2 -1347.257} C_VEL
LIN {X 0,Y 587.387,Z 347.317,A -85,B 0,C 180,E1 -1350,E2 -1350} C_VEL
LIN {X 0,Y 587.371,Z 347.317,A -85,B 0,C 180,E1 -1352.743,E2 -1352.743} C_VEL
LIN {X 0,Y 587.366,Z 347.324,A -85,B 0,C 180,E1 -1355.493,E2 -1355.493} C_VEL
LIN {X 0,Y 587.369,Z 347.319,A -85,B 0,C 180,E1 -1358.255,E2 -1358.255} C_VEL
LIN {X 0,Y 587.353,Z 347.319,A -85,B 0,C 180,E1 -1361.134,E2 -1361.134} C_VEL
LIN {X 0,Y 587.369,Z 347.318,A -85,B 0,C 180,E1 -1364.26,E2 -1364.26} C_VEL
LIN {X 0,Y 587.354,Z 347.322,A -85,B 0,C 180,E1 -1367.406,E2 -1367.406} C_VEL
LIN {X 0,Y 587.334,Z 347.327,A -85,B 0,C 180,E1 -1370.305,E2 -1370.305} C_VEL
LIN {X 0,Y 587.325,Z 347.324,A -85,B 0,C 180,E1 -1373.259,E2 -1373.259} C_VEL
LIN {X 0,Y 587.338,Z 347.327,A -85,B 0,C 180,E1 -1375.517,E2 -1375.517} C_VEL
LIN {X 0,Y 587.352,Z 347.319,A -85,B 0,C 180,E1 -1377.818,E2 -1377.818} C_VEL
LIN {X 0,Y 587.338,Z 347.328,A -85,B 0,C 180,E1 -1380.51,E2 -1380.51} C_VEL
LIN {X 0,Y 587.34,Z 347.323,A -85,B 0,C 180,E1 -1383.397,E2 -1383.397} C_VEL
LIN {X 0,Y 587.294,Z 347.328,A -85,B 0,C 180,E1 -1385.9,E2 -1385.9} C_VEL
LIN {X 0,Y 587.332,Z 347.325,A -85,B 0,C 180,E1 -1388.479,E2 -1388.479} C_VEL
LIN {X 0,Y 587.341,Z 347.321,A -85,B 0,C 180,E1 -1391.157,E2 -1391.157} C_VEL
LIN {X 0,Y 587.339,Z 347.324,A -85,B 0,C 180,E1 -1394.114,E2 -1394.114} C_VEL
LIN {X 0,Y 587.315,Z 347.329,A -85,B 0,C 180,E1 -1396.993,E2 -1396.993} C_VEL
LIN {X 0,Y 587.32,Z 347.323,A -85,B 0,C 180,E1 -1399.746,E2 -1399.746} C_VEL
LIN {X 0,Y 587.347,Z 347.324,A -85,B 0,C 180,E1 -1402.392,E2 -1402.392} C_VEL
LIN {X 0,Y 587.333,Z 347.322,A -85,B 0,C 180,E1 -1404.945,E2 -1404.945} C_VEL
LIN {X 0,Y 587.338,Z 347.325,A -85,B 0,C 180,E1 -1407.421,E2 -1407.421} C_VEL
LIN {X 0,Y 587.34,Z 347.342,A -85,B 0,C 180,E1 -1410.226,E2 -1410.226} C_VEL
LIN {X 0,Y 587.322,Z 353.882,A -85,B 0,C 180,E1 -1412.953,E2 -1412.953} C_VEL
LIN {X 0,Y 587.283,Z 359.616,A -85,B 0,C 180,E1 -1415.436,E2 -1415.436} C_VEL
LIN {X 0,Y 587.242,Z 366.326,A -85,B 0,C 180,E1 -1418.222,E2 -1418.222} C_VEL
LIN {X 0,Y 587.242,Z 373.542,A -85,B 0,C 180,E1 -1421.148,E2 -1421.148} C_VEL
LIN {X 0,Y 587.22,Z 380.758,A -85,B 0,C 180,E1 -1424.022,E2 -1424.022} C_VEL
LIN {X 0,Y 587.177,Z 387.974,A -85,B 0,C 180,E1 -1426.855,E2 -1426.855} C_VEL
LIN {X 0,Y 587.138,Z 395.191,A -85,B 0,C 180,E1 -1429.656,E2 -1429.656} C_VEL
LIN {X 0,Y 587.145,Z 402.408,A -85,B 0,C 180,E1 -1432.434,E2 -1432.434} C_VEL
LIN {X 0,Y 587.174,Z 403.705,A -85,B 0,C 180,E1 -1432.931,E2 -1432.931} C_VEL
LIN {X 0,Y 587.356,Z 412.472,A -85,B 0,C 180,E1 -1433.228,E2 -1433.228} C_VEL
LIN {X 0,Y 587.312,Z 420.815,A -85,B 0,C 180,E1 -1433.633,E2 -1433.633} C_VEL
LIN {X 0,Y 587.25,Z 429.02,A -85,B 0,C 180,E1 -1434.161,E2 -1434.161} C_VEL
LIN {X 0,Y 587.254,Z 437.042,A -85,B 0,C 180,E1 -1434.85,E2 -1434.85} C_VEL
LIN {X 0,Y 587.216,Z 443.218,A -85,B 0,C 180,E1 -1435.538,E2 -1435.538} C_VEL
LIN {X 0,Y 587.228,Z 448.077,A -85,B 0,C 180,E1 -1436.226,E2 -1436.226} C_VEL
LIN {X 0,Y 587.183,Z 451.826,A -85,B 0,C 180,E1 -1436.913,E2 -1436.913} C_VEL
LIN {X 0,Y 587.145,Z 455.832,A -85,B 0,C 180,E1 -1437.942,E2 -1437.942} C_VEL
LIN {X 0,Y 587.149,Z 457.574,A -85,B 0,C 180,E1 -1438.628,E2 -1438.628} C_VEL
LIN {X 0,Y 587.14,Z 458.618,A -85,B 0,C 180,E1 -1439.314,E2 -1439.314} C_VEL
LIN {X 0,Y 587.137,Z 458.996,A -85,B 0,C 180,E1 -1440,E2 -1440} C_VEL
LIN {X 0,Y 587.14,Z 458.713,A -85,B 0,C 180,E1 -1440.686,E2 -1440.686} C_VEL
LIN {X 0,Y 587.148,Z 457.765,A -85,B 0,C 180,E1 -1441.372,E2 -1441.372} C_VEL
LIN {X 0,Y 587.144,Z 456.124,A -85,B 0,C 180,E1 -1442.058,E2 -1442.058} C_VEL
LIN {X 0,Y 587.145,Z 453.739,A -85,B 0,C 180,E1 -1442.744,E2 -1442.744} C_VEL
LIN {X 0,Y 587.228,Z 448.609,A -85,B 0,C 180,E1 -1443.774,E2 -1443.774} C_VEL
LIN {X 0,Y 587.246,Z 442.542,A -85,B 0,C 180,E1 -1444.634,E2 -1444.634} C_VEL
LIN {X 0,Y 587.191,Z 436.231,A -85,B 0,C 180,E1 -1445.322,E2 -1445.322} C_VEL
LIN {X 0,Y 587.249,Z 429.075,A -85,B 0,C 180,E1 -1445.925,E2 -1445.925} C_VEL
LIN {X 0,Y 587.284,Z 420.299,A -85,B 0,C 180,E1 -1446.487,E2 -1446.487} C_VEL
LIN {X 0,Y 587.367,Z 411.049,A -85,B 0,C 180,E1 -1446.915,E2 -1446.915} C_VEL
LIN {X 0,Y 587.159,Z 403.658,A -85,B 0,C 180,E1 -1447.177,E2 -1447.177} C_VEL
LIN {X 0,Y 587.175,Z 397.229,A -85,B 0,C 180,E1 -1449.647,E2 -1449.647} C_VEL
LIN {X 0,Y 587.164,Z 390.01,A -85,B 0,C 180,E1 -1452.442,E2 -1452.442} C_VEL
LIN {X 0,Y 587.208,Z 384.595,A -85,B 0,C 180,E1 -1454.557,E2 -1454.557} C_VEL
LIN {X 0,Y 587.221,Z 377.376,A -85,B 0,C 180,E1 -1457.41,E2 -1457.41} C_VEL
LIN {X 0,Y 587.22,Z 371.961,A -85,B 0,C 180,E1 -1459.579,E2 -1459.579} C_VEL
LIN {X 0,Y 587.257,Z 364.741,A -85,B 0,C 180,E1 -1462.517,E2 -1462.517} C_VEL
LIN {X 0,Y 587.296,Z 359.469,A -85,B 0,C 180,E1 -1464.761,E2 -1464.761} C_VEL
LIN {X 0,Y 587.326,Z 354.121,A -85,B 0,C 180,E1 -1467.046,E2 -1467.046} C_VEL
LIN {X 0,Y 587.354,Z 347.324,A -85,B 0,C 180,E1 -1469.872,E2 -1469.872} C_VEL
LIN {X 0,Y 587.341,Z 347.327,A -85,B 0,C 180,E1 -1472.579,E2 -1472.579} C_VEL
LIN {X 0,Y 587.332,Z 347.327,A -85,B 0,C 180,E1 -1475.055,E2 -1475.055} C_VEL
LIN {X 0,Y 587.344,Z 347.327,A -85,B 0,C 180,E1 -1477.839,E2 -1477.839} C_VEL
LIN {X 0,Y 587.323,Z 347.329,A -85,B 0,C 180,E1 -1480.254,E2 -1480.254} C_VEL
LIN {X 0,Y 587.325,Z 347.328,A -85,B 0,C 180,E1 -1483.006,E2 -1483.006} C_VEL
LIN {X 0,Y 587.339,Z 347.325,A -85,B 0,C 180,E1 -1485.886,E2 -1485.886} C_VEL
LIN {X 0,Y 587.34,Z 347.325,A -85,B 0,C 180,E1 -1488.925,E2 -1488.925} C_VEL
LIN {X 0,Y 587.324,Z 347.329,A -85,B 0,C 180,E1 -1491.52,E2 -1491.52} C_VEL
LIN {X 0,Y 587.295,Z 347.331,A -85,B 0,C 180,E1 -1494.1,E2 -1494.1} C_VEL
LIN {X 0,Y 587.34,Z 347.327,A -85,B 0,C 180,E1 -1496.603,E2 -1496.603} C_VEL
LIN {X 0,Y 587.341,Z 347.326,A -85,B 0,C 180,E1 -1499.49,E2 -1499.49} C_VEL
LIN {X 0,Y 587.381,Z 347.481,A -85,B 0,C 180,E1 -1501.747,E2 -1501.747} C_VEL
LIN {X 0,Y 588.042,Z 350.599,A -85,B 0,C 180,E1 -1502.331,E2 -1502.331} C_VEL
LIN {X 0,Y 587.883,Z 367.206,A -85,B 0,C 180,E1 -1505.076,E2 -1505.076} C_VEL
LIN {X 0,Y 587.742,Z 384.515,A -85,B 0,C 180,E1 -1507.873,E2 -1507.873} C_VEL
LIN {X 0,Y 587.618,Z 402.491,A -85,B 0,C 180,E1 -1510.721,E2 -1510.721} C_VEL
LIN {X 0,Y 587.487,Z 421.44,A -85,B 0,C 180,E1 -1513.672,E2 -1513.672} C_VEL
LIN {X 0,Y 587.399,Z 441.056,A -85,B 0,C 180,E1 -1516.684,E2 -1516.684} C_VEL
LIN {X 0,Y 587.364,Z 448.19,A -85,B 0,C 180,E1 -1517.749,E2 -1517.749} C_VEL
LIN {X 0,Y 587.727,Z 453.601,A -85,B 0,C 180,E1 -1517.833,E2 -1517.833} C_VEL
LIN {X 0,Y 587.69,Z 466.69,A -85,B 0,C 180,E1 -1518.117,E2 -1518.117} C_VEL
LIN {X 0,Y 587.639,Z 479.858,A -85,B 0,C 180,E1 -1518.555,E2 -1518.555} C_VEL
LIN {X 0,Y 587.556,Z 492.628,A -85,B 0,C 180,E1 -1519.141,E2 -1519.141} C_VEL
LIN {X 0,Y 587.467,Z 504.199,A -85,B 0,C 180,E1 -1519.836,E2 -1519.836} C_VEL
LIN {X 0,Y 587.367,Z 514.595,A -85,B 0,C 180,E1 -1520.617,E2 -1520.617} C_VEL
LIN {X 0,Y 587.322,Z 523.111,A -85,B 0,C 180,E1 -1521.397,E2 -1521.397} C_VEL
LIN {X 0,Y 587.274,Z 530.959,A -85,B 0,C 180,E1 -1522.263,E2 -1522.263} C_VEL
LIN {X 0,Y 587.23,Z 537.468,A -85,B 0,C 180,E1 -1523.126,E2 -1523.126} C_VEL
LIN {X 0,Y 587.236,Z 543.866,A -85,B 0,C 180,E1 -1524.161,E2 -1524.161} C_VEL
LIN {X 0,Y 587.147,Z 548.949,A -85,B 0,C 180,E1 -1525.194,E2 -1525.194} C_VEL
LIN {X 0,Y 587.212,Z 552.895,A -85,B 0,C 180,E1 -1526.226,E2 -1526.226} C_VEL
LIN {X 0,Y 587.132,Z 555.808,A -85,B 0,C 180,E1 -1527.255,E2 -1527.255} C_VEL
LIN {X 0,Y 587.141,Z 557.2,A -85,B 0,C 180,E1 -1527.942,E2 -1527.942} C_VEL
LIN {X 0,Y 587.14,Z 558.784,A -85,B 0,C 180,E1 -1529.314,E2 -1529.314} C_VEL
LIN {X 0,Y 587.137,Z 559,A -85,B 0,C 180,E1 -1530,E2 -1530} C_VEL
LIN {X 0,Y 587.147,Z 558.185,A -85,B 0,C 180,E1 -1531.372,E2 -1531.372} C_VEL
LIN {X 0,Y 587.141,Z 557.201,A -85,B 0,C 180,E1 -1532.058,E2 -1532.058} C_VEL
LIN {X 0,Y 587.132,Z 555.81,A -85,B 0,C 180,E1 -1532.744,E2 -1532.744} C_VEL
LIN {X 0,Y 587.212,Z 552.897,A -85,B 0,C 180,E1 -1533.774,E2 -1533.774} C_VEL
LIN {X 0,Y 587.147,Z 548.95,A -85,B 0,C 180,E1 -1534.806,E2 -1534.806} C_VEL
LIN {X 0,Y 587.217,Z 542.879,A -85,B 0,C 180,E1 -1536.011,E2 -1536.011} C_VEL
LIN {X 0,Y 587.245,Z 536.238,A -85,B 0,C 180,E1 -1537.046,E2 -1537.046} C_VEL
LIN {X 0,Y 587.299,Z 527.991,A -85,B 0,C 180,E1 -1538.083,E2 -1538.083} C_VEL
LIN {X 0,Y 587.343,Z 519.538,A -85,B 0,C 180,E1 -1538.949,E2 -1538.949} C_VEL
LIN {X 0,Y 587.422,Z 509.096,A -85,B 0,C 180,E1 -1539.816,E2 -1539.816} C_VEL
LIN {X 0,Y 587.488,Z 498.76,A -85,B 0,C 180,E1 -1540.511,E2 -1540.511} C_VEL
LIN {X 0,Y 587.583,Z 486.812,A -85,B 0,C 180,E1 -1541.149,E2 -1541.149} C_VEL
LIN {X 0,Y 587.63,Z 474.598,A -85,B 0,C 180,E1 -1541.639,E2 -1541.639} C_VEL
LIN {X 0,Y 587.679,Z 461.44,A -85,B 0,C 180,E1 -1542.014,E2 -1542.014} C_VEL
LIN {X 0,Y 587.517,Z 449.29,A -85,B 0,C 180,E1 -1542.234,E2 -1542.234} C_VEL
LIN {X 0,Y 587.347,Z 447.982,A -85,B 0,C 180,E1 -1542.262,E2 -1542.262} C_VEL
LIN {X 0,Y 587.451,Z 429.519,A -85,B 0,C 180,E1 -1545.082,E2 -1545.082} C_VEL
LIN {X 0,Y 587.541,Z 412.21,A -85,B 0,C 180,E1 -1547.76,E2 -1547.76} C_VEL
LIN {X 0,Y 587.657,Z 394.902,A -85,B 0,C 180,E1 -1550.476,E2 -1550.476} C_VEL
LIN {X 0,Y 587.78,Z 377.593,A -85,B 0,C 180,E1 -1553.239,E2 -1553.239} C_VEL
LIN {X 0,Y 587.963,Z 360.284,A -85,B 0,C 180,E1 -1556.058,E2 -1556.058} C_VEL
LIN {X 0,Y 587.88,Z 349.908,A -85,B 0,C 180,E1 -1557.79,E2 -1557.79} C_VEL
LIN {X 0,Y 587.369,Z 347.322,A -85,B 0,C 180,E1 -1558.278,E2 -1558.278} C_VEL
LIN {X 0,Y 587.332,Z 347.323,A -85,B 0,C 180,E1 -1560.966,E2 -1560.966} C_VEL
LIN {X 0,Y 587.338,Z 347.327,A -85,B 0,C 180,E1 -1563.396,E2 -1563.396} C_VEL
LIN {X 0,Y 587.294,Z 347.327,A -85,B 0,C 180,E1 -1565.9,E2 -1565.9} C_VEL
LIN {X 0,Y 587.329,Z 347.329,A -85,B 0,C 180,E1 -1568.479,E2 -1568.479} C_VEL
LIN {X 0,Y 587.339,Z 347.321,A -85,B 0,C 180,E1 -1571.157,E2 -1571.157} C_VEL
LIN {X 0,Y 587.337,Z 347.322,A -85,B 0,C 180,E1 -1574.114,E2 -1574.114} C_VEL
LIN {X 0,Y 587.323,Z 347.328,A -85,B 0,C 180,E1 -1576.994,E2 -1576.994} C_VEL
LIN {X 0,Y 587.318,Z 347.325,A -85,B 0,C 180,E1 -1579.746,E2 -1579.746} C_VEL
LIN {X 0,Y 587.347,Z 347.321,A -85,B 0,C 180,E1 -1582.392,E2 -1582.392} C_VEL
LIN {X 0,Y 587.333,Z 347.326,A -85,B 0,C 180,E1 -1584.945,E2 -1584.945} C_VEL
LIN {X 0,Y 587.339,Z 347.322,A -85,B 0,C 180,E1 -1587.421,E2 -1587.421} C_VEL
LIN {X 0,Y 587.337,Z 347.323,A -85,B 0,C 180,E1 -1589.83,E2 -1589.83} C_VEL
LIN {X 0,Y 587.354,Z 347.321,A -85,B 0,C 180,E1 -1592.307,E2 -1592.307} C_VEL
LIN {X 0,Y 587.353,Z 347.326,A -85,B 0,C 180,E1 -1595.241,E2 -1595.241} C_VEL
LIN {X 0,Y 587.325,Z 347.326,A -85,B 0,C 180,E1 -1598.226,E2 -1598.226} C_VEL
LIN {X 0,Y 587.348,Z 347.32,A -85,B 0,C 180,E1 -1601.151,E2 -1601.151} C_VEL
LIN {X 0,Y 587.327,Z 347.324,A -85,B 0,C 180,E1 -1604.025,E2 -1604.025} C_VEL
LIN {X 0,Y 587.363,Z 347.318,A -85,B 0,C 180,E1 -1606.154,E2 -1606.154} C_VEL
LIN {X 0,Y 587.341,Z 347.323,A -85,B 0,C 180,E1 -1608.962,E2 -1608.962} C_VEL
LIN {X 0,Y 587.366,Z 347.322,A -85,B 0,C 180,E1 -1611.745,E2 -1611.745} C_VEL
LIN {X 0,Y 587.357,Z 347.318,A -85,B 0,C 180,E1 -1614.507,E2 -1614.507} C_VEL
LIN {X 0,Y 587.38,Z 347.318,A -85,B 0,C 180,E1 -1617.257,E2 -1617.257} C_VEL
LIN {X 0,Y 587.386,Z 347.319,A -85,B 0,C 180,E1 -1620,E2 -1620} C_VEL
LIN {X 0,Y 587.376,Z 347.316,A -85,B 0,C 180,E1 -1622.743,E2 -1622.743} C_VEL
LIN {X 0,Y 587.362,Z 347.322,A -85,B 0,C 180,E1 -1625.493,E2 -1625.493} C_VEL
LIN {X 0,Y 587.371,Z 347.32,A -85,B 0,C 180,E1 -1628.255,E2 -1628.255} C_VEL
LIN {X 0,Y 587.35,Z 347.319,A -85,B 0,C 180,E1 -1631.134,E2 -1631.134} C_VEL
LIN {X 0,Y 587.367,Z 347.317,A -85,B 0,C 180,E1 -1634.26,E2 -1634.26} C_VEL
LIN {X 0,Y 587.352,Z 347.321,A -85,B 0,C 180,E1 -1637.406,E2 -1637.406} C_VEL
LIN {X 0,Y 587.314,Z 347.325,A -85,B 0,C 180,E1 -1638.312,E2 -1638.312} C_VEL
LIN {X 0,Y 586.671,Z 347.408,A -85,B 0,C 180,E1 -1638.884,E2 -1638.884} C_VEL
LIN {X 0,Y 583.846,Z 347.758,A -85,B 0,C 180,E1 -1639.813,E2 -1639.813} C_VEL
LIN {X 0,Y 581.434,Z 348.06,A -85,B 0,C 180,E1 -1640.56,E2 -1640.56} C_VEL
LIN {X 0,Y 580.38,Z 348.189,A -85,B 0,C 180,E1 -1641.136,E2 -1641.136} C_VEL
LIN {X 0,Y 580.285,Z 348.2,A -85,B 0,C 180,E1 -1641.331,E2 -1641.331} C_VEL
LIN {X 0,Y 580.303,Z 348.197,A -85,B 0,C 180,E1 -1644.316,E2 -1644.316} C_VEL
LIN {X 0,Y 580.279,Z 348.203,A -85,B 0,C 180,E1 -1646.623,E2 -1646.623} C_VEL
LIN {X 0,Y 580.304,Z 348.198,A -85,B 0,C 180,E1 -1649.31,E2 -1649.31} C_VEL
LIN {X 0,Y 580.298,Z 348.202,A -85,B 0,C 180,E1 -1652.201,E2 -1652.201} C_VEL
LIN {X 0,Y 580.297,Z 348.199,A -85,B 0,C 180,E1 -1654.696,E2 -1654.696} C_VEL
LIN {X 0,Y 580.3,Z 348.201,A -85,B 0,C 180,E1 -1657.269,E2 -1657.269} C_VEL
LIN {X 0,Y 580.299,Z 348.204,A -85,B 0,C 180,E1 -1660.271,E2 -1660.271} C_VEL
LIN {X 0,Y 580.279,Z 348.201,A -85,B 0,C 180,E1 -1662.706,E2 -1662.706} C_VEL
LIN {X 0,Y 580.277,Z 348.204,A -85,B 0,C 180,E1 -1665.609,E2 -1665.609} C_VEL
LIN {X 0,Y 580.316,Z 348.197,A -85,B 0,C 180,E1 -1668.234,E2 -1668.234} C_VEL
LIN {X 0,Y 580.281,Z 348.201,A -85,B 0,C 180,E1 -1670.965,E2 -1670.965} C_VEL
LIN {X 0,Y 580.27,Z 348.208,A -85,B 0,C 180,E1 -1673.597,E2 -1673.597} C_VEL
LIN {X 0,Y 580.319,Z 348.195,A -85,B 0,C 180,E1 -1676.146,E2 -1676.146} C_VEL
LIN {X 0,Y 580.28,Z 348.207,A -85,B 0,C 180,E1 -1678.615,E2 -1678.615} C_VEL
LIN {X 0,Y 580.296,Z 348.198,A -85,B 0,C 180,E1 -1681.024,E2 -1681.024} C_VEL
LIN {X 0,Y 580.295,Z 348.205,A -85,B 0,C 180,E1 -1683.666,E2 -1683.666} C_VEL
LIN {X 0,Y 580.303,Z 348.2,A -85,B 0,C 180,E1 -1685.684,E2 -1685.684} C_VEL
LIN {X 0,Y 580.275,Z 348.201,A -85,B 0,C 180,E1 -1687.948,E2 -1687.948} C_VEL
LIN {X 0,Y 580.304,Z 348.198,A -85,B 0,C 180,E1 -1690.914,E2 -1690.914} C_VEL
LIN {X 0,Y 580.283,Z 348.206,A -85,B 0,C 180,E1 -1693.826,E2 -1693.826} C_VEL
LIN {X 0,Y 580.33,Z 348.195,A -85,B 0,C 180,E1 -1695.983,E2 -1695.983} C_VEL
LIN {X 0,Y 580.309,Z 348.202,A -85,B 0,C 180,E1 -1698.827,E2 -1698.827} C_VEL
LIN {X 0,Y 580.33,Z 348.196,A -85,B 0,C 180,E1 -1701.644,E2 -1701.644} C_VEL
LIN {X 0,Y 580.33,Z 348.194,A -85,B 0,C 180,E1 -1704.44,E2 -1704.44} C_VEL
LIN {X 0,Y 580.346,Z 348.192,A -85,B 0,C 180,E1 -1707.918,E2 -1707.918} C_VEL
LIN {X 0,Y 580.365,Z 348.193,A -85,B 0,C 180,E1 -1710.694,E2 -1710.694} C_VEL
LIN {X 0,Y 580.283,Z 348.203,A -85,B 0,C 180,E1 -1713.472,E2 -1713.472} C_VEL
LIN {X 0,Y 580.333,Z 348.199,A -85,B 0,C 180,E1 -1715.56,E2 -1715.56} C_VEL
LIN {X 0,Y 580.332,Z 348.196,A -85,B 0,C 180,E1 -1718.356,E2 -1718.356} C_VEL
LIN {X 0,Y 580.305,Z 348.197,A -85,B 0,C 180,E1 -1721.191,E2 -1721.191} C_VEL
LIN {X 0,Y 580.329,Z 348.197,A -85,B 0,C 180,E1 -1724.017,E2 -1724.017} C_VEL
LIN {X 0,Y 580.317,Z 348.2,A -85,B 0,C 180,E1 -1726.914,E2 -1726.914} C_VEL
LIN {X 0,Y 580.293,Z 348.199,A -85,B 0,C 180,E1 -1729.823,E2 -1729.823} C_VEL
LIN {X 0,Y 580.278,Z 348.207,A -85,B 0,C 180,E1 -1732.053,E2 -1732.053} C_VEL
LIN {X 0,Y 580.311,Z 348.198,A -85,B 0,C 180,E1 -1735.08,E2 -1735.08} C_VEL
LIN {X 0,Y 580.304,Z 348.198,A -85,B 0,C 180,E1 -1738.186,E2 -1738.186} C_VEL
LIN {X 0,Y 580.286,Z 348.203,A -85,B 0,C 180,E1 -1740.694,E2 -1740.694} C_VEL
LIN {X 0,Y 580.309,Z 348.198,A -85,B 0,C 180,E1 -1743.317,E2 -1743.317} C_VEL
LIN {X 0,Y 580.249,Z 348.207,A -85,B 0,C 180,E1 -1745.756,E2 -1745.756} C_VEL
LIN {X 0,Y 580.291,Z 348.199,A -85,B 0,C 180,E1 -1748.146,E2 -1748.146} C_VEL
LIN {X 0,Y 580.302,Z 348.2,A -85,B 0,C 180,E1 -1750.843,E2 -1750.843} C_VEL
LIN {X 0,Y 580.292,Z 348.204,A -85,B 0,C 180,E1 -1753.657,E2 -1753.657} C_VEL
LIN {X 0,Y 580.277,Z 348.201,A -85,B 0,C 180,E1 -1756.61,E2 -1756.61} C_VEL
LIN {X 0,Y 580.302,Z 348.2,A -85,B 0,C 180,E1 -1759.157,E2 -1759.157} C_VEL
LIN {X 0,Y 580.294,Z 348.203,A -85,B 0,C 180,E1 -1761.927,E2 -1761.927} C_VEL
LIN {X 0,Y 580.291,Z 348.199,A -85,B 0,C 180,E1 -1764.455,E2 -1764.455} C_VEL
LIN {X 0,Y 580.292,Z 348.203,A -85,B 0,C 180,E1 -1766.975,E2 -1766.975} C_VEL
LIN {X 0,Y 580.32,Z 348.198,A -85,B 0,C 180,E1 -1770.129,E2 -1770.129} C_VEL
LIN {X 0,Y 580.256,Z 352.816,A -85,B 0,C 180,E1 -1772.15,E2 -1772.15} C_VEL
LIN {X 0,Y 580.244,Z 359.278,A -85,B 0,C 180,E1 -1774.917,E2 -1774.917} C_VEL
LIN {X 0,Y 580.191,Z 366.328,A -85,B 0,C 180,E1 -1777.944,E2 -1777.944} C_VEL
LIN {X 0,Y 580.184,Z 373.544,A -85,B 0,C 180,E1 -1780.909,E2 -1780.909} C_VEL
LIN {X 0,Y 580.148,Z 380.759,A -85,B 0,C 180,E1 -1783.822,E2 -1783.822} C_VEL
LIN {X 0,Y 580.091,Z 387.976,A -85,B 0,C 180,E1 -1786.692,E2 -1786.692} C_VEL
LIN {X 0,Y 580.058,Z 395.192,A -85,B 0,C 180,E1 -1789.529,E2 -1789.529} C_VEL
LIN {X 0,Y 580.068,Z 402.409,A -85,B 0,C 180,E1 -1792.341,E2 -1792.341} C_VEL
LIN {X 0,Y 580.073,Z 403.706,A -85,B 0,C 180,E1 -1792.844,E2 -1792.844} C_VEL
LIN {X 0,Y 580.312,Z 411.516,A -85,B 0,C 180,E1 -1793.108,E2 -1793.108} C_VEL
LIN {X 0,Y 580.252,Z 420.792,A -85,B 0,C 180,E1 -1793.554,E2 -1793.554} C_VEL
LIN {X 0,Y 580.188,Z 429.029,A -85,B 0,C 180,E1 -1794.09,E2 -1794.09} C_VEL
LIN {X 0,Y 580.183,Z 437.047,A -85,B 0,C 180,E1 -1794.787,E2 -1794.787} C_VEL
LIN {X 0,Y 580.151,Z 443.222,A -85,B 0,C 180,E1 -1795.484,E2 -1795.484} C_VEL
LIN {X 0,Y 580.157,Z 448.081,A -85,B 0,C 180,E1 -1796.18,E2 -1796.18} C_VEL
LIN {X 0,Y 580.095,Z 451.829,A -85,B 0,C 180,E1 -1796.875,E2 -1796.875} C_VEL
LIN {X 0,Y 580.047,Z 455.834,A -85,B 0,C 180,E1 -1797.917,E2 -1797.917} C_VEL
LIN {X 0,Y 580.048,Z 457.575,A -85,B 0,C 180,E1 -1798.611,E2 -1798.611} C_VEL
LIN {X 0,Y 580.041,Z 458.619,A -85,B 0,C 180,E1 -1799.306,E2 -1799.306} C_VEL
LIN {X 0,Y 580.038,Z 458.996,A -85,B 0,C 180,E1 -1800,E2 -1800} C_VEL
LIN {X 0,Y 580.04,Z 458.712,A -85,B 0,C 180,E1 -1800.694,E2 -1800.694} C_VEL
LIN {X 0,Y 580.048,Z 457.763,A -85,B 0,C 180,E1 -1801.389,E2 -1801.389} C_VEL
LIN {X 0,Y 580.046,Z 456.123,A -85,B 0,C 180,E1 -1802.083,E2 -1802.083} C_VEL
LIN {X 0,Y 580.057,Z 453.737,A -85,B 0,C 180,E1 -1802.778,E2 -1802.778} C_VEL
LIN {X 0,Y 580.158,Z 448.607,A -85,B 0,C 180,E1 -1803.82,E2 -1803.82} C_VEL
LIN {X 0,Y 580.18,Z 442.537,A -85,B 0,C 180,E1 -1804.69,E2 -1804.69} C_VEL
LIN {X 0,Y 580.117,Z 436.225,A -85,B 0,C 180,E1 -1805.387,E2 -1805.387} C_VEL
LIN {X 0,Y 580.202,Z 429.069,A -85,B 0,C 180,E1 -1805.997,E2 -1805.997} C_VEL
LIN {X 0,Y 580.235,Z 421.282,A -85,B 0,C 180,E1 -1806.508,E2 -1806.508} C_VEL
LIN {X 0,Y 580.334,Z 412.206,A -85,B 0,C 180,E1 -1806.956,E2 -1806.956} C_VEL
LIN {X 0,Y 580.056,Z 403.656,A -85,B 0,C 180,E1 -1807.265,E2 -1807.265} C_VEL
LIN {X 0,Y 580.075,Z 397.227,A -85,B 0,C 180,E1 -1809.766,E2 -1809.766} C_VEL
LIN {X 0,Y 580.082,Z 390.008,A -85,B 0,C 180,E1 -1812.596,E2 -1812.596} C_VEL
LIN {X 0,Y 580.124,Z 384.594,A -85,B 0,C 180,E1 -1814.739,E2 -1814.739} C_VEL
LIN {X 0,Y 580.149,Z 377.375,A -85,B 0,C 180,E1 -1817.629,E2 -1817.629} C_VEL
LIN {X 0,Y 580.161,Z 371.96,A -85,B 0,C 180,E1 -1819.828,E2 -1819.828} C_VEL
LIN {X 0,Y 580.193,Z 366.545,A -85,B 0,C 180,E1 -1822.056,E2 -1822.056} C_VEL
LIN {X 0,Y 580.274,Z 359.826,A -85,B 0,C 180,E1 -1825.081,E2 -1825.081} C_VEL
LIN {X 0,Y 580.264,Z 354.114,A -85,B 0,C 180,E1 -1827.403,E2 -1827.403} C_VEL
LIN {X 0,Y 580.327,Z 348.2,A -85,B 0,C 180,E1 -1829.871,E2 -1829.871} C_VEL
LIN {X 0,Y 580.294,Z 348.204,A -85,B 0,C 180,E1 -1833.025,E2 -1833.025} C_VEL
LIN {X 0,Y 580.251,Z 348.21,A -85,B 0,C 180,E1 -1835.756,E2 -1835.756} C_VEL
LIN {X 0,Y 580.293,Z 348.205,A -85,B 0,C 180,E1 -1838.146,E2 -1838.146} C_VEL
LIN {X 0,Y 580.305,Z 348.202,A -85,B 0,C 180,E1 -1840.843,E2 -1840.843} C_VEL
LIN {X 0,Y 580.292,Z 348.203,A -85,B 0,C 180,E1 -1843.657,E2 -1843.657} C_VEL
LIN {X 0,Y 580.289,Z 348.205,A -85,B 0,C 180,E1 -1846.608,E2 -1846.608} C_VEL
LIN {X 0,Y 580.302,Z 348.202,A -85,B 0,C 180,E1 -1849.157,E2 -1849.157} C_VEL
LIN {X 0,Y 580.291,Z 348.204,A -85,B 0,C 180,E1 -1851.927,E2 -1851.927} C_VEL
LIN {X 0,Y 580.256,Z 348.208,A -85,B 0,C 180,E1 -1854.453,E2 -1854.453} C_VEL
LIN {X 0,Y 580.297,Z 348.206,A -85,B 0,C 180,E1 -1856.975,E2 -1856.975} C_VEL
LIN {X 0,Y 580.3,Z 348.203,A -85,B 0,C 180,E1 -1859.425,E2 -1859.425} C_VEL
LIN {X 0,Y 580.307,Z 348.228,A -85,B 0,C 180,E1 -1861.47,E2 -1861.47} C_VEL
LIN {X 0,Y 581.232,Z 352.933,A -85,B 0,C 180,E1 -1862.34,E2 -1862.34} C_VEL
LIN {X 0,Y 580.986,Z 368.36,A -85,B 0,C 180,E1 -1864.951,E2 -1864.951} C_VEL
LIN {X 0,Y 580.812,Z 385.669,A -85,B 0,C 180,E1 -1867.782,E2 -1867.782} C_VEL
LIN {X 0,Y 580.641,Z 404.202,A -85,B 0,C 180,E1 -1870.753,E2 -1870.753} C_VEL
LIN {X 0,Y 580.497,Z 422.594,A -85,B 0,C 180,E1 -1873.651,E2 -1873.651} C_VEL
LIN {X 0,Y 580.368,Z 441.056,A -85,B 0,C 180,E1 -1876.52,E2 -1876.52} C_VEL
LIN {X 0,Y 580.328,Z 448.19,A -85,B 0,C 180,E1 -1877.598,E2 -1877.598} C_VEL
LIN {X 0,Y 580.799,Z 453.6,A -85,B 0,C 180,E1 -1877.686,E2 -1877.686} C_VEL
LIN {X 0,Y 580.764,Z 466.69,A -85,B 0,C 180,E1 -1877.973,E2 -1877.973} C_VEL
LIN {X 0,Y 580.673,Z 479.171,A -85,B 0,C 180,E1 -1878.389,E2 -1878.389} C_VEL
LIN {X 0,Y 580.566,Z 490.925,A -85,B 0,C 180,E1 -1878.92,E2 -1878.92} C_VEL
LIN {X 0,Y 580.479,Z 501.581,A -85,B 0,C 180,E1 -1879.536,E2 -1879.536} C_VEL
LIN {X 0,Y 580.38,Z 512.472,A -85,B 0,C 180,E1 -1880.327,E2 -1880.327} C_VEL
LIN {X 0,Y 580.271,Z 523.111,A -85,B 0,C 180,E1 -1881.292,E2 -1881.292} C_VEL
LIN {X 0,Y 580.222,Z 530.959,A -85,B 0,C 180,E1 -1882.168,E2 -1882.168} C_VEL
LIN {X 0,Y 580.154,Z 538.649,A -85,B 0,C 180,E1 -1883.222,E2 -1883.222} C_VEL
LIN {X 0,Y 580.139,Z 545.679,A -85,B 0,C 180,E1 -1884.438,E2 -1884.438} C_VEL
LIN {X 0,Y 580.108,Z 550.371,A -85,B 0,C 180,E1 -1885.483,E2 -1885.483} C_VEL
LIN {X 0,Y 580.123,Z 553.956,A -85,B 0,C 180,E1 -1886.527,E2 -1886.527} C_VEL
LIN {X 0,Y 580.043,Z 555.808,A -85,B 0,C 180,E1 -1887.222,E2 -1887.222} C_VEL
LIN {X 0,Y 580.04,Z 557.199,A -85,B 0,C 180,E1 -1887.917,E2 -1887.917} C_VEL
LIN {X 0,Y 580.04,Z 558.784,A -85,B 0,C 180,E1 -1889.306,E2 -1889.306} C_VEL
LIN {X 0,Y 580.037,Z 559,A -85,B 0,C 180,E1 -1890,E2 -1890} C_VEL
LIN {X 0,Y 580.047,Z 558.185,A -85,B 0,C 180,E1 -1891.388,E2 -1891.388} C_VEL
LIN {X 0,Y 580.04,Z 557.201,A -85,B 0,C 180,E1 -1892.083,E2 -1892.083} C_VEL
LIN {X 0,Y 580.043,Z 555.81,A -85,B 0,C 180,E1 -1892.778,E2 -1892.778} C_VEL
LIN {X 0,Y 580.109,Z 552.897,A -85,B 0,C 180,E1 -1893.82,E2 -1893.82} C_VEL
LIN {X 0,Y 580.054,Z 548.95,A -85,B 0,C 180,E1 -1894.865,E2 -1894.865} C_VEL
LIN {X 0,Y 580.139,Z 542.878,A -85,B 0,C 180,E1 -1896.085,E2 -1896.085} C_VEL
LIN {X 0,Y 580.184,Z 536.238,A -85,B 0,C 180,E1 -1897.132,E2 -1897.132} C_VEL
LIN {X 0,Y 580.25,Z 527.992,A -85,B 0,C 180,E1 -1898.182,E2 -1898.182} C_VEL
LIN {X 0,Y 580.308,Z 519.539,A -85,B 0,C 180,E1 -1899.058,E2 -1899.058} C_VEL
LIN {X 0,Y 580.425,Z 509.097,A -85,B 0,C 180,E1 -1899.936,E2 -1899.936} C_VEL
LIN {X 0,Y 580.494,Z 498.758,A -85,B 0,C 180,E1 -1900.639,E2 -1900.639} C_VEL
LIN {X 0,Y 580.597,Z 487.243,A -85,B 0,C 180,E1 -1901.264,E2 -1901.264} C_VEL
LIN {X 0,Y 580.684,Z 474.474,A -85,B 0,C 180,E1 -1901.785,E2 -1901.785} C_VEL
LIN {X 0,Y 580.76,Z 461.439,A -85,B 0,C 180,E1 -1902.16,E2 -1902.16} C_VEL
LIN {X 0,Y 580.616,Z 450.232,A -85,B 0,C 180,E1 -1902.368,E2 -1902.368} C_VEL
LIN {X 0,Y 580.314,Z 447.982,A -85,B 0,C 180,E1 -1902.413,E2 -1902.413} C_VEL
LIN {X 0,Y 580.438,Z 430.673,A -85,B 0,C 180,E1 -1905.089,E2 -1905.089} C_VEL
LIN {X 0,Y 580.543,Z 413.364,A -85,B 0,C 180,E1 -1907.799,E2 -1907.799} C_VEL
LIN {X 0,Y 580.698,Z 396.056,A -85,B 0,C 180,E1 -1910.547,E2 -1910.547} C_VEL
LIN {X 0,Y 580.859,Z 379.128,A -85,B 0,C 180,E1 -1913.282,E2 -1913.282} C_VEL
LIN {X 0,Y 581.101,Z 361.609,A -85,B 0,C 180,E1 -1916.167,E2 -1916.167} C_VEL
LIN {X 0,Y 581.178,Z 352.796,A -85,B 0,C 180,E1 -1917.658,E2 -1917.658} C_VEL
LIN {X 0,Y 580.294,Z 348.206,A -85,B 0,C 180,E1 -1918.531,E2 -1918.531} C_VEL
LIN {X 0,Y 580.28,Z 348.203,A -85,B 0,C 180,E1 -1921.385,E2 -1921.385} C_VEL
LIN {X 0,Y 580.319,Z 348.198,A -85,B 0,C 180,E1 -1923.854,E2 -1923.854} C_VEL
LIN {X 0,Y 580.3,Z 348.203,A -85,B 0,C 180,E1 -1926.934,E2 -1926.934} C_VEL
LIN {X 0,Y 580.286,Z 348.203,A -85,B 0,C 180,E1 -1929.933,E2 -1929.933} C_VEL
LIN {X 0,Y 580.284,Z 348.2,A -85,B 0,C 180,E1 -1932.706,E2 -1932.706} C_VEL
LIN {X 0,Y 580.277,Z 348.203,A -85,B 0,C 180,E1 -1935.608,E2 -1935.608} C_VEL
LIN {X 0,Y 580.282,Z 348.203,A -85,B 0,C 180,E1 -1938.231,E2 -1938.231} C_VEL
LIN {X 0,Y 580.292,Z 348.198,A -85,B 0,C 180,E1 -1940.966,E2 -1940.966} C_VEL
LIN {X 0,Y 580.286,Z 348.206,A -85,B 0,C 180,E1 -1943.597,E2 -1943.597} C_VEL
LIN {X 0,Y 580.319,Z 348.196,A -85,B 0,C 180,E1 -1946.145,E2 -1946.145} C_VEL
LIN {X 0,Y 580.289,Z 348.205,A -85,B 0,C 180,E1 -1948.615,E2 -1948.615} C_VEL
LIN {X 0,Y 580.295,Z 348.198,A -85,B 0,C 180,E1 -1951.024,E2 -1951.024} C_VEL
LIN {X 0,Y 580.293,Z 348.204,A -85,B 0,C 180,E1 -1953.666,E2 -1953.666} C_VEL
LIN {X 0,Y 580.3,Z 348.199,A -85,B 0,C 180,E1 -1955.684,E2 -1955.684} C_VEL
LIN {X 0,Y 580.287,Z 348.204,A -85,B 0,C 180,E1 -1958.695,E2 -1958.695} C_VEL
LIN {X 0,Y 580.301,Z 348.198,A -85,B 0,C 180,E1 -1960.913,E2 -1960.913} C_VEL
LIN {X 0,Y 580.281,Z 348.203,A -85,B 0,C 180,E1 -1963.826,E2 -1963.826} C_VEL
LIN {X 0,Y 580.329,Z 348.194,A -85,B 0,C 180,E1 -1965.983,E2 -1965.983} C_VEL
LIN {X 0,Y 580.307,Z 348.201,A -85,B 0,C 180,E1 -1968.827,E2 -1968.827} C_VEL
LIN {X 0,Y 580.33,Z 348.198,A -85,B 0,C 180,E1 -1971.644,E2 -1971.644} C_VEL
LIN {X 0,Y 580.323,Z 348.195,A -85,B 0,C 180,E1 -1974.44,E2 -1974.44} C_VEL
LIN {X 0,Y 580.346,Z 348.195,A -85,B 0,C 180,E1 -1977.224,E2 -1977.224} C_VEL
LIN {X 0,Y 580.355,Z 348.195,A -85,B 0,C 180,E1 -1980,E2 -1980} C_VEL
LIN {X 0,Y 580.342,Z 348.192,A -85,B 0,C 180,E1 -1982.777,E2 -1982.777} C_VEL
LIN {X 0,Y 580.327,Z 348.197,A -85,B 0,C 180,E1 -1985.56,E2 -1985.56} C_VEL
LIN {X 0,Y 580.336,Z 348.197,A -85,B 0,C 180,E1 -1988.356,E2 -1988.356} C_VEL
LIN {X 0,Y 580.302,Z 348.198,A -85,B 0,C 180,E1 -1991.191,E2 -1991.191} C_VEL
LIN {X 0,Y 580.327,Z 348.196,A -85,B 0,C 180,E1 -1994.017,E2 -1994.017} C_VEL
LIN {X 0,Y 580.314,Z 348.202,A -85,B 0,C 180,E1 -1996.914,E2 -1996.914} C_VEL
LIN {X 0,Y 580.308,Z 348.198,A -85,B 0,C 180,E1 -1999.822,E2 -1999.822} C_VEL
LIN {X 0,Y 580.285,Z 348.2,A -85,B 0,C 180,E1 -2001.331,E2 -2001.331} C_VEL
LIN {X 0,Y 579.588,Z 348.293,A -85,B 0,C 180,E1 -2001.911,E2 -2001.911} C_VEL
LIN {X 0,Y 576.711,Z 348.646,A -85,B 0,C 180,E1 -2002.851,E2 -2002.851} C_VEL
LIN {X 0,Y 574.317,Z 348.95,A -85,B 0,C 180,E1 -2003.607,E2 -2003.607} C_VEL
LIN {X 0,Y 573.319,Z 349.069,A -85,B 0,C 180,E1 -2004.191,E2 -2004.191} C_VEL
LIN {X 0,Y 573.252,Z 349.076,A -85,B 0,C 180,E1 -2004.388,E2 -2004.388} C_VEL
LIN {X 0,Y 573.253,Z 349.083,A -85,B 0,C 180,E1 -2006.976,E2 -2006.976} C_VEL
LIN {X 0,Y 573.249,Z 349.076,A -85,B 0,C 180,E1 -2009.488,E2 -2009.488} C_VEL
LIN {X 0,Y 573.255,Z 349.076,A -85,B 0,C 180,E1 -2012.645,E2 -2012.645} C_VEL
LIN {X 0,Y 573.256,Z 349.081,A -85,B 0,C 180,E1 -2015.185,E2 -2015.185} C_VEL
LIN {X 0,Y 573.237,Z 349.077,A -85,B 0,C 180,E1 -2017.808,E2 -2017.808} C_VEL
LIN {X 0,Y 573.272,Z 349.078,A -85,B 0,C 180,E1 -2020.528,E2 -2020.528} C_VEL
LIN {X 0,Y 573.246,Z 349.083,A -85,B 0,C 180,E1 -2023.669,E2 -2023.669} C_VEL
LIN {X 0,Y 573.25,Z 349.078,A -85,B 0,C 180,E1 -2026.642,E2 -2026.642} C_VEL
LIN {X 0,Y 573.246,Z 349.076,A -85,B 0,C 180,E1 -2029.475,E2 -2029.475} C_VEL
LIN {X 0,Y 573.238,Z 349.082,A -85,B 0,C 180,E1 -2032.193,E2 -2032.193} C_VEL
LIN {X 0,Y 573.239,Z 349.083,A -85,B 0,C 180,E1 -2035.229,E2 -2035.229} C_VEL
LIN {X 0,Y 573.255,Z 349.075,A -85,B 0,C 180,E1 -2037.772,E2 -2037.772} C_VEL
LIN {X 0,Y 573.266,Z 349.077,A -85,B 0,C 180,E1 -2040.634,E2 -2040.634} C_VEL
LIN {X 0,Y 573.254,Z 349.076,A -85,B 0,C 180,E1 -2043.024,E2 -2043.024} C_VEL
LIN {X 0,Y 573.278,Z 349.079,A -85,B 0,C 180,E1 -2045.366,E2 -2045.366} C_VEL
LIN {X 0,Y 573.232,Z 349.082,A -85,B 0,C 180,E1 -2048.42,E2 -2048.42} C_VEL
LIN {X 0,Y 573.282,Z 349.074,A -85,B 0,C 180,E1 -2050.728,E2 -2050.728} C_VEL
LIN {X 0,Y 573.256,Z 349.081,A -85,B 0,C 180,E1 -2053.622,E2 -2053.622} C_VEL
LIN {X 0,Y 573.277,Z 349.075,A -85,B 0,C 180,E1 -2055.807,E2 -2055.807} C_VEL
LIN {X 0,Y 573.267,Z 349.08,A -85,B 0,C 180,E1 -2058.745,E2 -2058.745} C_VEL
LIN {X 0,Y 573.286,Z 349.072,A -85,B 0,C 180,E1 -2061.541,E2 -2061.541} C_VEL
LIN {X 0,Y 573.298,Z 349.07,A -85,B 0,C 180,E1 -2064.372,E2 -2064.372} C_VEL
LIN {X 0,Y 573.316,Z 349.068,A -85,B 0,C 180,E1 -2067.893,E2 -2067.893} C_VEL
LIN {X 0,Y 573.335,Z 349.068,A -85,B 0,C 180,E1 -2070.702,E2 -2070.702} C_VEL
LIN {X 0,Y 573.305,Z 349.069,A -85,B 0,C 180,E1 -2072.811,E2 -2072.811} C_VEL
LIN {X 0,Y 573.3,Z 349.074,A -85,B 0,C 180,E1 -2075.628,E2 -2075.628} C_VEL
LIN {X 0,Y 573.288,Z 349.075,A -85,B 0,C 180,E1 -2078.46,E2 -2078.46} C_VEL
LIN {X 0,Y 573.276,Z 349.073,A -85,B 0,C 180,E1 -2081.312,E2 -2081.312} C_VEL
LIN {X 0,Y 573.286,Z 349.071,A -85,B 0,C 180,E1 -2084.424,E2 -2084.424} C_VEL
LIN {X 0,Y 573.263,Z 349.081,A -85,B 0,C 180,E1 -2087.112,E2 -2087.112} C_VEL
LIN {X 0,Y 573.248,Z 349.079,A -85,B 0,C 180,E1 -2090.077,E2 -2090.077} C_VEL
LIN {X 0,Y 573.242,Z 349.081,A -85,B 0,C 180,E1 -2092.338,E2 -2092.338} C_VEL
LIN {X 0,Y 573.258,Z 349.081,A -85,B 0,C 180,E1 -2095.41,E2 -2095.41} C_VEL
LIN {X 0,Y 573.256,Z 349.075,A -85,B 0,C 180,E1 -2098.029,E2 -2098.029} C_VEL
LIN {X 0,Y 573.249,Z 349.08,A -85,B 0,C 180,E1 -2100.176,E2 -2100.176} C_VEL
LIN {X 0,Y 573.259,Z 349.076,A -85,B 0,C 180,E1 -2102.645,E2 -2102.645} C_VEL
LIN {X 0,Y 573.21,Z 349.084,A -85,B 0,C 180,E1 -2105.188,E2 -2105.188} C_VEL
LIN {X 0,Y 573.239,Z 349.078,A -85,B 0,C 180,E1 -2107.808,E2 -2107.808} C_VEL
LIN {X 0,Y 573.248,Z 349.083,A -85,B 0,C 180,E1 -2110.525,E2 -2110.525} C_VEL
LIN {X 0,Y 573.251,Z 349.078,A -85,B 0,C 180,E1 -2113.358,E2 -2113.358} C_VEL
LIN {X 0,Y 573.242,Z 349.077,A -85,B 0,C 180,E1 -2116.332,E2 -2116.332} C_VEL
LIN {X 0,Y 573.232,Z 349.081,A -85,B 0,C 180,E1 -2118.543,E2 -2118.543} C_VEL
LIN {X 0,Y 573.253,Z 349.076,A -85,B 0,C 180,E1 -2121.299,E2 -2121.299} C_VEL
LIN {X 0,Y 573.249,Z 349.081,A -85,B 0,C 180,E1 -2124.014,E2 -2124.014} C_VEL
LIN {X 0,Y 573.273,Z 349.073,A -85,B 0,C 180,E1 -2126.518,E2 -2126.518} C_VEL
LIN {X 0,Y 573.237,Z 349.082,A -85,B 0,C 180,E1 -2129.117,E2 -2129.117} C_VEL
LIN {X 0,Y 573.287,Z 349.114,A -85,B 0,C 180,E1 -2130.199,E2 -2130.199} C_VEL
LIN {X 0,Y 573.2,Z 355.78,A -85,B 0,C 180,E1 -2133.021,E2 -2133.021} C_VEL
LIN {X 0,Y 573.201,Z 361.152,A -85,B 0,C 180,E1 -2135.363,E2 -2135.363} C_VEL
LIN {X 0,Y 573.104,Z 368.185,A -85,B 0,C 180,E1 -2138.414,E2 -2138.414} C_VEL
LIN {X 0,Y 573.067,Z 375.349,A -85,B 0,C 180,E1 -2141.406,E2 -2141.406} C_VEL
LIN {X 0,Y 573.082,Z 380.761,A -85,B 0,C 180,E1 -2143.617,E2 -2143.617} C_VEL
LIN {X 0,Y 573.023,Z 387.977,A -85,B 0,C 180,E1 -2146.524,E2 -2146.524} C_VEL
LIN {X 0,Y 572.989,Z 395.194,A -85,B 0,C 180,E1 -2149.398,E2 -2149.398} C_VEL
LIN {X 0,Y 572.986,Z 403.313,A -85,B 0,C 180,E1 -2152.6,E2 -2152.6} C_VEL
LIN {X 0,Y 572.97,Z 403.707,A -85,B 0,C 180,E1 -2152.755,E2 -2152.755} C_VEL
LIN {X 0,Y 573.254,Z 409.773,A -85,B 0,C 180,E1 -2152.958,E2 -2152.958} C_VEL
LIN {X 0,Y 573.208,Z 418.558,A -85,B 0,C 180,E1 -2153.346,E2 -2153.346} C_VEL
LIN {X 0,Y 573.175,Z 426.593,A -85,B 0,C 180,E1 -2153.841,E2 -2153.841} C_VEL
LIN {X 0,Y 573.083,Z 433.316,A -85,B 0,C 180,E1 -2154.37,E2 -2154.37} C_VEL
LIN {X 0,Y 573.092,Z 440.378,A -85,B 0,C 180,E1 -2155.075,E2 -2155.075} C_VEL
LIN {X 0,Y 573.037,Z 445.767,A -85,B 0,C 180,E1 -2155.78,E2 -2155.78} C_VEL
LIN {X 0,Y 573.062,Z 450.029,A -85,B 0,C 180,E1 -2156.484,E2 -2156.484} C_VEL
LIN {X 0,Y 572.972,Z 453.346,A -85,B 0,C 180,E1 -2157.188,E2 -2157.188} C_VEL
LIN {X 0,Y 572.951,Z 455.836,A -85,B 0,C 180,E1 -2157.891,E2 -2157.891} C_VEL
LIN {X 0,Y 572.948,Z 457.577,A -85,B 0,C 180,E1 -2158.594,E2 -2158.594} C_VEL
LIN {X 0,Y 572.941,Z 458.62,A -85,B 0,C 180,E1 -2159.297,E2 -2159.297} C_VEL
LIN {X 0,Y 572.938,Z 458.996,A -85,B 0,C 180,E1 -2160,E2 -2160} C_VEL
LIN {X 0,Y 572.941,Z 458.711,A -85,B 0,C 180,E1 -2160.703,E2 -2160.703} C_VEL
LIN {X 0,Y 572.948,Z 457.762,A -85,B 0,C 180,E1 -2161.406,E2 -2161.406} C_VEL
LIN {X 0,Y 572.95,Z 456.121,A -85,B 0,C 180,E1 -2162.109,E2 -2162.109} C_VEL
LIN {X 0,Y 572.973,Z 453.734,A -85,B 0,C 180,E1 -2162.812,E2 -2162.812} C_VEL
LIN {X 0,Y 573.085,Z 448.604,A -85,B 0,C 180,E1 -2163.867,E2 -2163.867} C_VEL
LIN {X 0,Y 573.109,Z 442.533,A -85,B 0,C 180,E1 -2164.748,E2 -2164.748} C_VEL
LIN {X 0,Y 573.047,Z 436.218,A -85,B 0,C 180,E1 -2165.454,E2 -2165.454} C_VEL
LIN {X 0,Y 573.156,Z 429.063,A -85,B 0,C 180,E1 -2166.071,E2 -2166.071} C_VEL
LIN {X 0,Y 573.177,Z 421.271,A -85,B 0,C 180,E1 -2166.588,E2 -2166.588} C_VEL
LIN {X 0,Y 573.297,Z 412.193,A -85,B 0,C 180,E1 -2167.042,E2 -2167.042} C_VEL
LIN {X 0,Y 572.973,Z 403.655,A -85,B 0,C 180,E1 -2167.355,E2 -2167.355} C_VEL
LIN {X 0,Y 572.987,Z 397.226,A -85,B 0,C 180,E1 -2169.888,E2 -2169.888} C_VEL
LIN {X 0,Y 573.009,Z 391.812,A -85,B 0,C 180,E1 -2172.035,E2 -2172.035} C_VEL
LIN {X 0,Y 573.049,Z 384.592,A -85,B 0,C 180,E1 -2174.925,E2 -2174.925} C_VEL
LIN {X 0,Y 573.085,Z 377.373,A -85,B 0,C 180,E1 -2177.854,E2 -2177.854} C_VEL
LIN {X 0,Y 573.108,Z 370.188,A -85,B 0,C 180,E1 -2180.832,E2 -2180.832} C_VEL
LIN {X 0,Y 573.177,Z 365.106,A -85,B 0,C 180,E1 -2183.13,E2 -2183.13} C_VEL
LIN {X 0,Y 573.232,Z 359.832,A -85,B 0,C 180,E1 -2185.411,E2 -2185.411} C_VEL
LIN {X 0,Y 573.216,Z 353.521,A -85,B 0,C 180,E1 -2188.022,E2 -2188.022} C_VEL
LIN {X 0,Y 573.312,Z 349.074,A -85,B 0,C 180,E1 -2189.89,E2 -2189.89} C_VEL
LIN {X 0,Y 573.257,Z 349.082,A -85,B 0,C 180,E1 -2192.645,E2 -2192.645} C_VEL
LIN {X 0,Y 573.213,Z 349.086,A -85,B 0,C 180,E1 -2195.188,E2 -2195.188} C_VEL
LIN {X 0,Y 573.24,Z 349.083,A -85,B 0,C 180,E1 -2197.807,E2 -2197.807} C_VEL
LIN {X 0,Y 573.274,Z 349.078,A -85,B 0,C 180,E1 -2200.528,E2 -2200.528} C_VEL
LIN {X 0,Y 573.257,Z 349.08,A -85,B 0,C 180,E1 -2203.67,E2 -2203.67} C_VEL
LIN {X 0,Y 573.251,Z 349.081,A -85,B 0,C 180,E1 -2206.642,E2 -2206.642} C_VEL
LIN {X 0,Y 573.248,Z 349.083,A -85,B 0,C 180,E1 -2209.475,E2 -2209.475} C_VEL
LIN {X 0,Y 573.237,Z 349.082,A -85,B 0,C 180,E1 -2212.192,E2 -2212.192} C_VEL
LIN {X 0,Y 573.24,Z 349.082,A -85,B 0,C 180,E1 -2215.228,E2 -2215.228} C_VEL
LIN {X 0,Y 573.257,Z 349.082,A -85,B 0,C 180,E1 -2217.771,E2 -2217.771} C_VEL
LIN {X 0,Y 573.269,Z 349.08,A -85,B 0,C 180,E1 -2220.634,E2 -2220.634} C_VEL
LIN {X 0,Y 573.297,Z 349.205,A -85,B 0,C 180,E1 -2221.213,E2 -2221.213} C_VEL
LIN {X 0,Y 574.412,Z 354.834,A -85,B 0,C 180,E1 -2222.294,E2 -2222.294} C_VEL
LIN {X 0,Y 574.067,Z 370.267,A -85,B 0,C 180,E1 -2224.951,E2 -2224.951} C_VEL
LIN {X 0,Y 573.858,Z 387.976,A -85,B 0,C 180,E1 -2227.877,E2 -2227.877} C_VEL
LIN {X 0,Y 573.66,Z 405.285,A -85,B 0,C 180,E1 -2230.684,E2 -2230.684} C_VEL
LIN {X 0,Y 573.476,Z 423.748,A -85,B 0,C 180,E1 -2233.628,E2 -2233.628} C_VEL
LIN {X 0,Y 573.33,Z 441.056,A -85,B 0,C 180,E1 -2236.351,E2 -2236.351} C_VEL
LIN {X 0,Y 573.279,Z 448.078,A -85,B 0,C 180,E1 -2237.441,E2 -2237.441} C_VEL
LIN {X 0,Y 573.88,Z 453.6,A -85,B 0,C 180,E1 -2237.535,E2 -2237.535} C_VEL
LIN {X 0,Y 573.832,Z 466.689,A -85,B 0,C 180,E1 -2237.826,E2 -2237.826} C_VEL
LIN {X 0,Y 573.719,Z 479.913,A -85,B 0,C 180,E1 -2238.276,E2 -2238.276} C_VEL
LIN {X 0,Y 573.608,Z 492.626,A -85,B 0,C 180,E1 -2238.873,E2 -2238.873} C_VEL
LIN {X 0,Y 573.434,Z 504.2,A -85,B 0,C 180,E1 -2239.585,E2 -2239.585} C_VEL
LIN {X 0,Y 573.334,Z 514.598,A -85,B 0,C 180,E1 -2240.385,E2 -2240.385} C_VEL
LIN {X 0,Y 573.241,Z 523.111,A -85,B 0,C 180,E1 -2241.184,E2 -2241.184} C_VEL
LIN {X 0,Y 573.161,Z 530.959,A -85,B 0,C 180,E1 -2242.071,E2 -2242.071} C_VEL
LIN {X 0,Y 573.073,Z 538.58,A -85,B 0,C 180,E1 -2243.126,E2 -2243.126} C_VEL
LIN {X 0,Y 573.07,Z 545.679,A -85,B 0,C 180,E1 -2244.369,E2 -2244.369} C_VEL
LIN {X 0,Y 573.028,Z 550.371,A -85,B 0,C 180,E1 -2245.427,E2 -2245.427} C_VEL
LIN {X 0,Y 573.022,Z 553.957,A -85,B 0,C 180,E1 -2246.484,E2 -2246.484} C_VEL
LIN {X 0,Y 572.959,Z 555.808,A -85,B 0,C 180,E1 -2247.188,E2 -2247.188} C_VEL
LIN {X 0,Y 572.94,Z 557.198,A -85,B 0,C 180,E1 -2247.891,E2 -2247.891} C_VEL
LIN {X 0,Y 572.941,Z 558.785,A -85,B 0,C 180,E1 -2249.297,E2 -2249.297} C_VEL
LIN {X 0,Y 572.938,Z 559,A -85,B 0,C 180,E1 -2250,E2 -2250} C_VEL
LIN {X 0,Y 572.946,Z 558.186,A -85,B 0,C 180,E1 -2251.406,E2 -2251.406} C_VEL
LIN {X 0,Y 572.939,Z 557.2,A -85,B 0,C 180,E1 -2252.109,E2 -2252.109} C_VEL
LIN {X 0,Y 572.959,Z 555.81,A -85,B 0,C 180,E1 -2252.812,E2 -2252.812} C_VEL
LIN {X 0,Y 573.014,Z 552.897,A -85,B 0,C 180,E1 -2253.868,E2 -2253.868} C_VEL
LIN {X 0,Y 572.963,Z 548.95,A -85,B 0,C 180,E1 -2254.925,E2 -2254.925} C_VEL
LIN {X 0,Y 573.064,Z 542.878,A -85,B 0,C 180,E1 -2256.16,E2 -2256.16} C_VEL
LIN {X 0,Y 573.119,Z 536.239,A -85,B 0,C 180,E1 -2257.221,E2 -2257.221} C_VEL
LIN {X 0,Y 573.201,Z 527.992,A -85,B 0,C 180,E1 -2258.283,E2 -2258.283} C_VEL
LIN {X 0,Y 573.287,Z 519.539,A -85,B 0,C 180,E1 -2259.17,E2 -2259.17} C_VEL
LIN {X 0,Y 573.43,Z 509.098,A -85,B 0,C 180,E1 -2260.058,E2 -2260.058} C_VEL
LIN {X 0,Y 573.51,Z 498.776,A -85,B 0,C 180,E1 -2260.769,E2 -2260.769} C_VEL
LIN {X 0,Y 573.628,Z 487.59,A -85,B 0,C 180,E1 -2261.385,E2 -2261.385} C_VEL
LIN {X 0,Y 573.729,Z 475.77,A -85,B 0,C 180,E1 -2261.885,E2 -2261.885} C_VEL
LIN {X 0,Y 573.814,Z 462.352,A -85,B 0,C 180,E1 -2262.287,E2 -2262.287} C_VEL
LIN {X 0,Y 573.714,Z 451.079,A -85,B 0,C 180,E1 -2262.507,E2 -2262.507} C_VEL
LIN {X 0,Y 573.261,Z 447.982,A -85,B 0,C 180,E1 -2262.569,E2 -2262.569} C_VEL
LIN {X 0,Y 573.408,Z 430.673,A -85,B 0,C 180,E1 -2265.279,E2 -2265.279} C_VEL
LIN {X 0,Y 573.551,Z 414.518,A -85,B 0,C 180,E1 -2267.839,E2 -2267.839} C_VEL
LIN {X 0,Y 573.757,Z 397.209,A -85,B 0,C 180,E1 -2270.619,E2 -2270.619} C_VEL
LIN {X 0,Y 573.954,Z 380.743,A -85,B 0,C 180,E1 -2273.311,E2 -2273.311} C_VEL
LIN {X 0,Y 574.245,Z 362.187,A -85,B 0,C 180,E1 -2276.417,E2 -2276.417} C_VEL
LIN {X 0,Y 574.335,Z 354.642,A -85,B 0,C 180,E1 -2277.71,E2 -2277.71} C_VEL
LIN {X 0,Y 573.276,Z 349.079,A -85,B 0,C 180,E1 -2278.762,E2 -2278.762} C_VEL
LIN {X 0,Y 573.245,Z 349.083,A -85,B 0,C 180,E1 -2281.815,E2 -2281.815} C_VEL
LIN {X 0,Y 573.27,Z 349.074,A -85,B 0,C 180,E1 -2284.328,E2 -2284.328} C_VEL
LIN {X 0,Y 573.253,Z 349.078,A -85,B 0,C 180,E1 -2287.166,E2 -2287.166} C_VEL
LIN {X 0,Y 573.241,Z 349.078,A -85,B 0,C 180,E1 -2289.607,E2 -2289.607} C_VEL
LIN {X 0,Y 573.246,Z 349.077,A -85,B 0,C 180,E1 -2292.642,E2 -2292.642} C_VEL
LIN {X 0,Y 573.242,Z 349.078,A -85,B 0,C 180,E1 -2295.667,E2 -2295.667} C_VEL
LIN {X 0,Y 573.232,Z 349.085,A -85,B 0,C 180,E1 -2298.543,E2 -2298.543} C_VEL
LIN {X 0,Y 573.251,Z 349.076,A -85,B 0,C 180,E1 -2301.299,E2 -2301.299} C_VEL
LIN {X 0,Y 573.248,Z 349.078,A -85,B 0,C 180,E1 -2304.014,E2 -2304.014} C_VEL
LIN {X 0,Y 573.271,Z 349.076,A -85,B 0,C 180,E1 -2306.518,E2 -2306.518} C_VEL
LIN {X 0,Y 573.24,Z 349.078,A -85,B 0,C 180,E1 -2309.116,E2 -2309.116} C_VEL
LIN {X 0,Y 573.255,Z 349.081,A -85,B 0,C 180,E1 -2311.971,E2 -2311.971} C_VEL
LIN {X 0,Y 573.255,Z 349.076,A -85,B 0,C 180,E1 -2314.59,E2 -2314.59} C_VEL
LIN {X 0,Y 573.237,Z 349.078,A -85,B 0,C 180,E1 -2317.662,E2 -2317.662} C_VEL
LIN {X 0,Y 573.28,Z 349.073,A -85,B 0,C 180,E1 -2320.728,E2 -2320.728} C_VEL
LIN {X 0,Y 573.254,Z 349.082,A -85,B 0,C 180,E1 -2323.622,E2 -2323.622} C_VEL
LIN {X 0,Y 573.276,Z 349.074,A -85,B 0,C 180,E1 -2325.807,E2 -2325.807} C_VEL
LIN {X 0,Y 573.265,Z 349.079,A -85,B 0,C 180,E1 -2328.745,E2 -2328.745} C_VEL
LIN {X 0,Y 573.286,Z 349.074,A -85,B 0,C 180,E1 -2331.541,E2 -2331.541} C_VEL
LIN {X 0,Y 573.29,Z 349.071,A -85,B 0,C 180,E1 -2334.372,E2 -2334.372} C_VEL
LIN {X 0,Y 573.312,Z 349.072,A -85,B 0,C 180,E1 -2337.189,E2 -2337.189} C_VEL
LIN {X 0,Y 573.325,Z 349.071,A -85,B 0,C 180,E1 -2340,E2 -2340} C_VEL
LIN {X 0,Y 573.308,Z 349.069,A -85,B 0,C 180,E1 -2342.811,E2 -2342.811} C_VEL
LIN {X 0,Y 573.293,Z 349.073,A -85,B 0,C 180,E1 -2345.628,E2 -2345.628} C_VEL
LIN {X 0,Y 573.292,Z 349.076,A -85,B 0,C 180,E1 -2348.459,E2 -2348.459} C_VEL
LIN {X 0,Y 573.274,Z 349.074,A -85,B 0,C 180,E1 -2351.312,E2 -2351.312} C_VEL
LIN {X 0,Y 573.283,Z 349.072,A -85,B 0,C 180,E1 -2354.424,E2 -2354.424} C_VEL
LIN {X 0,Y 573.261,Z 349.079,A -85,B 0,C 180,E1 -2357.112,E2 -2357.112} C_VEL
LIN {X 0,Y 573.255,Z 349.08,A -85,B 0,C 180,E1 -2360.077,E2 -2360.077} C_VEL
LIN {X 0,Y 573.236,Z 349.079,A -85,B 0,C 180,E1 -2363.099,E2 -2363.099} C_VEL
LIN {X 0,Y 573.252,Z 349.076,A -85,B 0,C 180,E1 -2364.388,E2 -2364.388} C_VEL
LIN {X 0,Y 572.626,Z 349.158,A -85,B 0,C 180,E1 -2364.975,E2 -2364.975} C_VEL
LIN {X 0,Y 569.783,Z 349.511,A -85,B 0,C 180,E1 -2365.926,E2 -2365.926} C_VEL
LIN {X 0,Y 567.351,Z 349.815,A -85,B 0,C 180,E1 -2366.691,E2 -2366.691} C_VEL
LIN {X 0,Y 566.295,Z 349.945,A -85,B 0,C 180,E1 -2367.283,E2 -2367.283} C_VEL
LIN {X 0,Y 566.205,Z 349.954,A -85,B 0,C 180,E1 -2367.483,E2 -2367.483} C_VEL
LIN {X 0,Y 566.203,Z 349.955,A -85,B 0,C 180,E1 -2369.769,E2 -2369.769} C_VEL
LIN {X 0,Y 566.205,Z 349.955,A -85,B 0,C 180,E1 -2372.43,E2 -2372.43} C_VEL
LIN {X 0,Y 566.206,Z 349.956,A -85,B 0,C 180,E1 -2374.993,E2 -2374.993} C_VEL
LIN {X 0,Y 566.198,Z 349.955,A -85,B 0,C 180,E1 -2377.461,E2 -2377.461} C_VEL
LIN {X 0,Y 566.22,Z 349.957,A -85,B 0,C 180,E1 -2380.198,E2 -2380.198} C_VEL
LIN {X 0,Y 566.203,Z 349.955,A -85,B 0,C 180,E1 -2383.054,E2 -2383.054} C_VEL
LIN {X 0,Y 566.205,Z 349.954,A -85,B 0,C 180,E1 -2386.048,E2 -2386.048} C_VEL
LIN {X 0,Y 566.185,Z 349.96,A -85,B 0,C 180,E1 -2388.861,E2 -2388.861} C_VEL
LIN {X 0,Y 566.189,Z 349.958,A -85,B 0,C 180,E1 -2391.637,E2 -2391.637} C_VEL
LIN {X 0,Y 566.165,Z 349.959,A -85,B 0,C 180,E1 -2394.308,E2 -2394.308} C_VEL
